C09113=1137.061,-43.555,-47.132,179.183,6.181,149.357
C09114=1137.056,-43.306,-47.143,179.186,6.182,149.356
C09115=1137.051,-43.056,-47.155,179.188,6.183,149.355
C09116=1137.046,-42.806,-47.166,179.191,6.183,149.355
C09117=1137.041,-42.556,-47.177,179.193,6.184,149.354
C09118=1137.035,-42.307,-47.188,179.195,6.184,149.354
C09119=1137.030,-42.057,-47.199,179.198,6.185,149.353
C09120=1137.025,-41.807,-47.211,179.200,6.186,149.353
C09121=1137.020,-41.558,-47.222,179.202,6.186,149.352
C09122=1137.014,-41.308,-47.233,179.205,6.187,149.352
C09123=1137.009,-41.058,-47.245,179.207,6.188,149.351
C09124=1137.004,-40.808,-47.256,179.209,6.189,149.351
C09125=1136.998,-40.559,-47.267,179.212,6.189,149.350
C09126=1136.994,-40.309,-47.279,179.214,6.190,149.350
C09127=1136.988,-40.060,-47.291,179.216,6.191,149.349
C09128=1136.984,-39.810,-47.302,179.219,6.191,149.348
C09129=1136.977,-39.560,-47.313,179.221,6.192,149.348
C09130=1136.973,-39.310,-47.324,179.223,6.193,149.347
C09131=1136.967,-39.060,-47.336,179.226,6.193,149.347
C09132=1136.962,-38.811,-47.347,179.228,6.194,149.346
C09133=1136.956,-38.562,-47.359,179.230,6.195,149.346
C09134=1136.952,-38.312,-47.370,179.233,6.195,149.345
C09135=1136.946,-38.062,-47.382,179.235,6.196,149.345
C09136=1136.942,-37.812,-47.393,179.237,6.196,149.344
C09137=1136.936,-37.563,-47.405,179.239,6.196,149.343
C09138=1136.930,-37.313,-47.416,179.241,6.197,149.343
C09139=1136.925,-37.063,-47.427,179.244,6.198,149.342
C09140=1136.920,-36.813,-47.439,179.246,6.198,149.342
C09141=1136.915,-36.563,-47.450,179.248,6.199,149.341
C09142=1136.909,-36.314,-47.462,179.251,6.200,149.341
C09143=1136.904,-36.065,-47.473,179.253,6.200,149.340
C09144=1136.899,-35.815,-47.485,179.255,6.201,149.340
C09145=1136.893,-35.565,-47.497,179.258,6.202,149.339
C09146=1136.889,-35.315,-47.508,179.260,6.202,149.339
C09147=1136.883,-35.066,-47.520,179.263,6.203,149.338
C09148=1136.878,-34.816,-47.531,179.265,6.204,149.337
C09149=1136.873,-34.566,-47.543,179.267,6.204,149.337
C09150=1136.868,-34.317,-47.554,179.270,6.205,149.336
C09151=1136.862,-34.067,-47.566,179.272,6.206,149.336
C09152=1136.857,-33.817,-47.578,179.274,6.206,149.335
C09153=1136.852,-33.568,-47.589,179.277,6.207,149.335
C09154=1136.847,-33.319,-47.601,179.279,6.208,149.334
C09155=1136.841,-33.069,-47.613,179.281,6.208,149.334
C09156=1136.836,-32.819,-47.625,179.284,6.209,149.333
C09157=1136.831,-32.569,-47.637,179.286,6.210,149.333
C09158=1136.826,-32.319,-47.648,179.288,6.210,149.332
C09159=1136.821,-32.069,-47.660,179.291,6.211,149.331
C09160=1136.815,-31.820,-47.671,179.293,6.212,149.331
C09161=1136.810,-31.571,-47.683,179.296,6.213,149.330
C09162=1136.805,-31.321,-47.694,179.298,6.213,149.330
C09163=1136.799,-31.071,-47.706,179.301,6.214,149.329
C09164=1136.794,-30.821,-47.719,179.303,6.215,149.329
C09165=1136.790,-30.572,-47.730,179.305,6.215,149.328
C09166=1136.784,-30.322,-47.742,179.308,6.216,149.328
C09167=1136.779,-30.072,-47.754,179.310,6.217,149.327
C09168=1136.773,-29.823,-47.765,179.312,6.217,149.326
C09169=1136.768,-29.573,-47.777,179.315,6.218,149.326
C09170=1136.763,-29.324,-47.789,179.317,6.219,149.325
C09171=1136.758,-29.074,-47.801,179.319,6.219,149.325
C09172=1136.753,-28.824,-47.813,179.322,6.220,149.324
C09173=1136.747,-28.574,-47.824,179.324,6.221,149.324
C09174=1136.742,-28.324,-47.836,179.326,6.221,149.323
C09175=1136.737,-28.075,-47.848,179.329,6.222,149.323
C09176=1136.732,-27.825,-47.860,179.331,6.223,149.322
C09177=1136.727,-27.575,-47.872,179.333,6.223,149.321
C09178=1136.721,-27.325,-47.884,179.336,6.224,149.321
C09179=1136.717,-27.076,-47.896,179.338,6.225,149.321
C09180=1136.711,-26.827,-47.908,179.341,6.225,149.320
C09181=1136.706,-26.577,-47.920,179.343,6.226,149.319
C09182=1136.701,-26.327,-47.932,179.345,6.227,149.319
C09183=1136.696,-26.078,-47.943,179.348,6.227,149.318
C09184=1136.690,-25.828,-47.955,179.350,6.228,149.318
C09185=1136.685,-25.579,-47.967,179.352,6.229,149.317
C09186=1136.680,-25.329,-47.980,179.355,6.230,149.317
C09187=1136.674,-25.059,-47.993,179.357,6.231,149.316
C09188=1136.669,-24.788,-48.006,179.360,6.231,149.315
C09189=1136.663,-24.519,-48.018,179.362,6.232,149.315
C09190=1136.657,-24.248,-48.032,179.365,6.232,149.314
C09191=1136.653,-23.999,-48.044,179.368,6.234,149.314
C09192=1136.647,-23.749,-48.056,179.370,6.235,149.313
C09193=1136.642,-23.499,-48.067,179.373,6.235,149.313
C09194=1136.637,-23.250,-48.080,179.375,6.236,149.312
C09195=1136.631,-23.000,-48.092,179.377,6.237,149.312
C09196=1136.626,-22.750,-48.104,179.380,6.237,149.311
C09197=1136.621,-22.501,-48.116,179.382,6.238,149.310
C09198=1136.616,-22.251,-48.128,179.384,6.238,149.310
C09199=1136.611,-22.002,-48.140,179.387,6.239,149.309
C09200=1136.605,-21.752,-48.152,179.389,6.240,149.309
C09201=1136.600,-21.503,-48.165,179.391,6.240,149.308
C09202=1136.595,-21.253,-48.177,179.394,6.241,149.308
C09203=1136.589,-21.003,-48.189,179.396,6.242,149.307
C09204=1136.584,-20.753,-48.201,179.399,6.243,149.306
C09205=1136.579,-20.503,-48.213,179.401,6.244,149.306
C09206=1136.574,-20.254,-48.226,179.403,6.245,149.306
C09207=1136.568,-20.004,-48.238,179.406,6.245,149.305
C09208=1136.563,-19.755,-48.250,179.408,6.246,149.304
C09209=1136.558,-19.505,-48.262,179.410,6.247,149.304
C09210=1136.553,-19.256,-48.275,179.413,6.247,149.303
C09211=1136.547,-19.006,-48.287,179.415,6.248,149.303
C09212=1136.543,-18.756,-48.299,179.417,6.249,149.302
C09213=1136.538,-18.507,-48.312,179.420,6.249,149.302
C09214=1136.533,-18.257,-48.323,179.422,6.250,149.301
C09215=1136.528,-18.007,-48.336,179.425,6.252,149.301
C09216=1136.522,-17.757,-48.348,179.428,6.252,149.300
C09217=1136.517,-17.508,-48.360,179.430,6.253,149.299
C09218=1136.512,-17.258,-48.372,179.432,6.254,149.299
C09219=1136.507,-17.009,-48.385,179.435,6.254,149.298
C09220=1136.501,-16.760,-48.398,179.437,6.255,149.298
C09221=1136.496,-16.510,-48.409,179.439,6.256,149.297
C09222=1136.491,-16.260,-48.422,179.442,6.256,149.297
C09223=1136.486,-16.010,-48.434,179.444,6.257,149.296
C09224=1136.481,-15.760,-48.447,179.447,6.258,149.296
C09225=1136.475,-15.511,-48.460,179.449,6.259,149.295
C09226=1136.470,-15.261,-48.472,179.452,6.259,149.295
C09227=1136.465,-15.011,-48.485,179.454,6.260,149.294
C09228=1136.459,-14.762,-48.497,179.456,6.261,149.293
C09229=1136.454,-14.512,-48.509,179.459,6.261,149.293
C09230=1136.449,-14.263,-48.522,179.461,6.262,149.292
C09231=1136.444,-14.013,-48.535,179.463,6.263,149.292
C09232=1136.439,-13.763,-48.547,179.466,6.264,149.291
C09233=1136.434,-13.514,-48.559,179.469,6.265,149.291
C09234=1136.429,-13.264,-48.572,179.471,6.265,149.290
C09235=1136.424,-13.015,-48.584,179.473,6.266,149.290
C09236=1136.418,-12.765,-48.596,179.476,6.267,149.289
C09237=1136.414,-12.515,-48.609,179.478,6.267,149.288
C09238=1136.408,-12.265,-48.622,179.480,6.268,149.288
C09239=1136.403,-12.016,-48.635,179.484,6.269,149.287
C09240=1136.397,-11.766,-48.647,179.486,6.270,149.287
C09241=1136.392,-11.517,-48.659,179.488,6.271,149.286
C09242=1136.388,-11.267,-48.672,179.491,6.271,149.286
C09243=1136.382,-11.018,-48.685,179.493,6.272,149.285
C09244=1136.377,-10.768,-48.698,179.495,6.273,149.285
C09245=1136.372,-10.518,-48.710,179.498,6.274,149.284
C09246=1136.366,-10.269,-48.723,179.500,6.275,149.284
C09247=1136.361,-10.019,-48.736,179.503,6.276,149.283
C09248=1136.356,-9.769,-48.748,179.505,6.276,149.282
C09249=1136.351,-9.520,-48.761,179.507,6.277,149.282
C09250=1136.346,-9.271,-48.773,179.510,6.278,149.281
C09251=1136.341,-9.020,-48.786,179.512,6.278,149.281
C09252=1136.335,-8.770,-48.799,179.515,6.280,149.280
C09253=1136.330,-8.521,-48.812,179.518,6.280,149.280
C09254=1136.325,-8.272,-48.824,179.520,6.281,149.279
C09255=1136.320,-8.022,-48.837,179.522,6.282,149.279
C09256=1136.316,-7.772,-48.850,179.525,6.282,149.278
C09257=1136.310,-7.523,-48.863,179.527,6.283,149.278
C09258=1136.305,-7.273,-48.876,179.530,6.285,149.277
C09259=1136.299,-7.024,-48.888,179.532,6.285,149.276
C09260=1136.295,-6.774,-48.901,179.534,6.286,149.276
C09261=1136.289,-6.524,-48.914,179.537,6.287,149.275
C09262=1136.284,-6.275,-48.926,179.539,6.287,149.275
C09263=1136.279,-6.025,-48.939,179.542,6.289,149.274
C09264=1136.274,-5.775,-48.952,179.544,6.290,149.274
C09265=1136.268,-5.526,-48.965,179.547,6.290,149.273
C09266=1136.263,-5.276,-48.978,179.549,6.291,149.273
C09267=1136.258,-5.026,-48.990,179.552,6.291,149.272
C09268=1136.253,-4.777,-49.004,179.554,6.292,149.272
C09269=1136.247,-4.527,-49.016,179.557,6.294,149.271
C09270=1136.243,-4.277,-49.029,179.559,6.294,149.270
C09271=1136.237,-4.028,-49.042,179.562,6.295,149.270
C09272=1136.232,-3.778,-49.055,179.564,6.296,149.269
C09273=1136.227,-3.528,-49.068,179.566,6.296,149.269
C09274=1136.222,-3.279,-49.082,179.569,6.298,149.268
C09275=1136.217,-3.030,-49.095,179.571,6.298,149.268
C09276=1136.212,-2.780,-49.107,179.574,6.299,149.267
C09277=1136.206,-2.530,-49.121,179.576,6.300,149.267
C09278=1136.201,-2.281,-49.133,179.578,6.300,149.266
C09279=1136.197,-2.031,-49.146,179.582,6.302,149.265
C09280=1136.191,-1.781,-49.159,179.584,6.302,149.265
C09281=1136.186,-1.532,-49.172,179.586,6.303,149.265
C09282=1136.181,-1.282,-49.185,179.589,6.304,149.264
C09283=1136.175,-1.032,-49.198,179.591,6.305,149.263
C09284=1136.171,-0.784,-49.212,179.594,6.306,149.263
C09285=1136.165,-0.533,-49.225,179.596,6.307,149.262
C09286=1136.160,-0.284,-49.238,179.598,6.307,149.262
C09287=1136.155,-0.035,-49.250,179.601,6.308,149.261
C09288=1136.150,0.216,-49.264,179.604,6.309,149.261
C09289=1136.145,0.465,-49.276,179.606,6.310,149.260
C09290=1136.140,0.715,-49.291,179.609,6.311,149.259
C09291=1136.134,0.984,-49.304,179.611,6.312,149.259
C09292=1136.128,1.254,-49.318,179.614,6.313,149.258
C09293=1136.123,1.523,-49.333,179.616,6.313,149.258
C09294=1136.117,1.792,-49.347,179.620,6.315,149.257
C09295=1136.112,2.042,-49.360,179.622,6.315,149.257
C09296=1136.107,2.291,-49.374,179.624,6.316,149.256
C09297=1136.102,2.541,-49.387,179.627,6.317,149.256
C09298=1136.097,2.791,-49.400,179.629,6.318,149.255
C09299=1136.091,3.040,-49.413,179.632,6.319,149.254
C09300=1136.087,3.290,-49.427,179.634,6.319,149.254
C09301=1136.081,3.539,-49.440,179.636,6.320,149.253
C09302=1136.076,3.789,-49.453,179.640,6.321,149.253
C09303=1136.071,4.038,-49.467,179.642,6.322,149.252
C09304=1136.066,4.288,-49.480,179.644,6.323,149.252
C09305=1136.060,4.538,-49.493,179.647,6.324,149.251
C09306=1136.056,4.787,-49.506,179.649,6.325,149.251
C09307=1136.050,5.037,-49.520,179.652,6.326,149.250
C09308=1136.045,5.286,-49.532,179.654,6.326,149.250
C09309=1136.040,5.536,-49.547,179.656,6.327,149.249
C09310=1136.035,5.785,-49.559,179.659,6.329,149.249
C09311=1136.030,6.036,-49.573,179.662,6.329,149.248
C09312=1136.024,6.285,-49.587,179.664,6.330,149.247
C09313=1136.020,6.535,-49.600,179.667,6.331,149.247
C09314=1136.014,6.784,-49.613,179.669,6.332,149.246
C09315=1136.010,7.034,-49.626,179.672,6.333,149.246
C09316=1136.004,7.283,-49.640,179.674,6.333,149.245
C09317=1136.000,7.533,-49.653,179.677,6.335,149.245
C09318=1135.994,7.782,-49.667,179.679,6.336,149.244
C09319=1135.989,8.032,-49.681,179.682,6.336,149.244
C09320=1135.984,8.282,-49.693,179.684,6.337,149.243
C09321=1135.979,8.531,-49.708,179.687,6.338,149.243
C09322=1135.973,8.781,-49.721,179.689,6.339,149.242
C09323=1135.969,9.030,-49.735,179.692,6.340,149.241
C09324=1135.963,9.280,-49.748,179.694,6.341,149.241
C09325=1135.959,9.529,-49.761,179.697,6.342,149.240
C09326=1135.953,9.780,-49.775,179.699,6.343,149.240
C09327=1135.948,10.029,-49.789,179.701,6.343,149.239
C09328=1135.943,10.279,-49.802,179.705,6.345,149.239
C09329=1135.938,10.528,-49.816,179.707,6.345,149.238
C09330=1135.932,10.778,-49.829,179.710,6.346,149.238
C09331=1135.928,11.027,-49.843,179.712,6.347,149.237
C09332=1135.922,11.277,-49.856,179.714,6.348,149.237
C09333=1135.917,11.526,-49.870,179.717,6.349,149.236
C09334=1135.912,11.776,-49.884,179.719,6.349,149.236
C09335=1135.907,12.026,-49.897,179.722,6.351,149.235
C09336=1135.902,12.275,-49.911,179.725,6.352,149.234
C09337=1135.897,12.525,-49.925,179.727,6.352,149.234
C09338=1135.892,12.774,-49.938,179.730,6.354,149.233
C09339=1135.887,13.024,-49.952,179.732,6.354,149.233
C09340=1135.881,13.273,-49.966,179.735,6.355,149.232
C09341=1135.876,13.523,-49.980,179.737,6.357,149.232
C09342=1135.872,13.772,-49.994,179.740,6.357,149.231
C09343=1135.866,14.022,-50.007,179.742,6.358,149.231
C09344=1135.861,14.272,-50.021,179.745,6.360,149.230
C09345=1135.856,14.521,-50.035,179.748,6.360,149.230
C09346=1135.851,14.771,-50.048,179.750,6.361,149.229
C09347=1135.846,15.020,-50.062,179.752,6.363,149.229
C09348=1135.840,15.269,-50.076,179.755,6.363,149.228
C09349=1135.835,15.520,-50.090,179.757,6.364,149.227
C09350=1135.830,15.769,-50.104,179.761,6.365,149.227
C09351=1135.825,16.018,-50.117,179.763,6.366,149.226
C09352=1135.820,16.268,-50.132,179.765,6.367,149.226
C09353=1135.815,16.518,-50.145,179.768,6.368,149.225
C09354=1135.809,16.767,-50.159,179.770,6.369,149.225
C09355=1135.805,17.017,-50.173,179.772,6.369,149.224
C09356=1135.800,17.267,-50.188,179.776,6.371,149.224
C09357=1135.794,17.516,-50.200,179.778,6.372,149.223
C09358=1135.790,17.766,-50.214,179.780,6.372,149.223
C09359=1135.785,18.015,-50.229,179.783,6.374,149.222
C09360=1135.779,18.264,-50.243,179.786,6.374,149.222
C09361=1135.774,18.514,-50.257,179.788,6.375,149.221
C09362=1135.769,18.764,-50.271,179.791,6.376,149.220
C09363=1135.763,19.013,-50.284,179.793,6.377,149.220
C09364=1135.758,19.263,-50.299,179.795,6.378,149.219
C09365=1135.754,19.512,-50.312,179.799,6.379,149.219
C09366=1135.749,19.761,-50.326,179.801,6.380,149.218
C09367=1135.744,20.011,-50.341,179.803,6.381,149.218
C09368=1135.739,20.261,-50.355,179.806,6.382,149.217
C09369=1135.734,20.511,-50.369,179.808,6.383,149.217
C09370=1135.728,20.760,-50.383,179.811,6.385,149.216
C09371=1135.723,21.009,-50.397,179.814,6.385,149.216
C09372=1135.718,21.260,-50.411,179.816,6.386,149.215
C09373=1135.713,21.509,-50.425,179.819,6.387,149.215
C09374=1135.707,21.758,-50.439,179.821,6.388,149.214
C09375=1135.702,22.008,-50.453,179.823,6.389,149.214
C09376=1135.697,22.258,-50.468,179.827,6.390,149.213
C09377=1135.692,22.508,-50.482,179.829,6.391,149.212
C09378=1135.687,22.757,-50.496,179.831,6.392,149.212
C09379=1135.682,23.006,-50.510,179.834,6.393,149.211
C09380=1135.677,23.256,-50.524,179.836,6.394,149.211
C09381=1135.672,23.506,-50.539,179.839,6.395,149.210
C09382=1135.667,23.755,-50.553,179.842,6.396,149.210
C09383=1135.662,24.004,-50.567,179.844,6.396,149.209
C09384=1135.657,24.254,-50.581,179.847,6.398,149.209
C09385=1135.652,24.504,-50.595,179.849,6.399,149.208
C09386=1135.647,24.753,-50.610,179.852,6.400,149.208
C09387=1135.641,25.002,-50.624,179.854,6.401,149.207
C09388=1135.636,25.252,-50.639,179.857,6.401,149.206
C09389=1135.632,25.501,-50.653,179.860,6.403,149.206
C09390=1135.627,25.751,-50.667,179.862,6.404,149.206
C09391=1135.622,26.001,-50.681,179.865,6.405,149.205
C09392=1135.616,26.250,-50.695,179.867,6.406,149.204
C09393=1135.611,26.499,-50.710,179.870,6.407,149.204
C09394=1135.606,26.749,-50.724,179.873,6.408,149.203
C09395=1135.600,27.018,-50.740,179.875,6.409,149.203
C09396=1135.595,27.288,-50.755,179.878,6.410,149.202
C09397=1135.590,27.556,-50.771,179.881,6.412,149.202
C09398=1135.584,27.825,-50.786,179.884,6.412,149.201
C09399=1135.579,28.074,-50.800,179.886,6.414,149.201
C09400=1135.574,28.324,-50.815,179.889,6.415,149.200
C09401=1135.568,28.574,-50.830,179.891,6.415,149.199
C09402=1135.563,28.824,-50.844,179.894,6.417,149.199
C09403=1135.559,29.073,-50.859,179.896,6.417,149.199
C09404=1135.554,29.323,-50.873,179.899,6.419,149.198
C09405=1135.549,29.572,-50.887,179.902,6.419,149.197
C09406=1135.543,29.821,-50.901,179.904,6.421,149.197
C09407=1135.538,30.071,-50.917,179.907,6.422,149.196
C09408=1135.533,30.320,-50.931,179.909,6.422,149.196
C09409=1135.528,30.570,-50.946,179.912,6.424,149.195
C09410=1135.523,30.820,-50.960,179.915,6.424,149.195
C09411=1135.518,31.069,-50.975,179.917,6.426,149.194
C09412=1135.513,31.319,-50.989,179.920,6.427,149.194
C09413=1135.508,31.569,-51.004,179.923,6.428,149.193
C09414=1135.503,31.818,-51.019,179.925,6.429,149.193
C09415=1135.498,32.067,-51.033,179.927,6.430,149.192
C09416=1135.493,32.316,-51.047,179.930,6.431,149.192
C09417=1135.487,32.566,-51.063,179.933,6.432,149.191
C09418=1135.482,32.816,-51.077,179.935,6.433,149.191
C09419=1135.477,33.065,-51.091,179.938,6.434,149.190
C09420=1135.473,33.314,-51.106,179.941,6.435,149.189
C09421=1135.467,33.564,-51.121,179.943,6.436,149.189
C09422=1135.462,33.813,-51.136,179.946,6.438,149.188
C09423=1135.457,34.063,-51.150,179.948,6.438,149.188
C09424=1135.452,34.313,-51.165,179.951,6.440,149.187
C09425=1135.447,34.562,-51.180,179.954,6.440,149.187
C09426=1135.442,34.812,-51.195,179.956,6.441,149.186
C09427=1135.437,35.061,-51.210,179.959,6.443,149.186
C09428=1135.432,35.311,-51.224,179.961,6.443,149.185
C09429=1135.427,35.560,-51.239,179.964,6.445,149.185
C09430=1135.422,35.810,-51.254,179.966,6.446,149.184
C09431=1135.417,36.059,-51.269,179.969,6.447,149.184
C09432=1135.412,36.309,-51.284,179.972,6.448,149.183
C09433=1135.407,36.558,-51.299,179.974,6.449,149.183
C09434=1135.401,36.808,-51.313,179.977,6.450,149.182
C09435=1135.397,37.057,-51.328,179.980,6.452,149.182
C09436=1135.392,37.307,-51.343,179.982,6.452,149.181
C09437=1135.386,37.556,-51.358,179.985,6.454,149.180
C09438=1135.382,37.806,-51.373,179.987,6.454,149.180
C09439=1135.376,38.055,-51.388,179.990,6.456,149.180
C09440=1135.371,38.305,-51.402,179.993,6.457,149.179
C09441=1135.367,38.554,-51.417,179.996,6.458,149.178
C09442=1135.361,38.804,-51.432,179.998,6.459,149.178
C09443=1135.356,39.053,-51.447,-180.000,6.461,149.178
C09444=1135.351,39.303,-51.463,-179.997,6.461,149.177
C09445=1135.346,39.552,-51.477,-179.994,6.463,149.176
C09446=1135.340,39.802,-51.493,-179.992,6.464,149.176
C09447=1135.335,40.052,-51.507,-179.989,6.465,149.175
C09448=1135.331,40.301,-51.522,-179.987,6.466,149.175
C09449=1135.325,40.550,-51.538,-179.984,6.467,149.174
C09450=1135.321,40.800,-51.552,-179.981,6.468,149.174
C09451=1135.315,41.049,-51.567,-179.978,6.469,149.173
C09452=1135.311,41.299,-51.583,-179.976,6.470,149.173
C09453=1135.305,41.549,-51.598,-179.973,6.471,149.172
C09454=1135.301,41.798,-51.613,-179.971,6.472,149.172
C09455=1135.295,42.047,-51.628,-179.968,6.474,149.171
C09456=1135.291,42.297,-51.643,-179.965,6.474,149.171
C09457=1135.285,42.547,-51.658,-179.963,6.476,149.170
C09458=1135.280,42.796,-51.673,-179.960,6.477,149.170
C09459=1135.275,43.045,-51.689,-179.958,6.478,149.169
C09460=1135.270,43.294,-51.704,-179.955,6.479,149.169
C09461=1135.265,43.545,-51.719,-179.952,6.480,149.168
C09462=1135.261,43.794,-51.734,-179.950,6.481,149.168
C09463=1135.255,44.043,-51.749,-179.947,6.483,149.167
C09464=1135.251,44.292,-51.764,-179.945,6.483,149.167
C09465=1135.245,44.542,-51.779,-179.942,6.485,149.166
C09466=1135.239,44.792,-51.795,-179.939,6.485,149.165
C09467=1135.235,45.041,-51.810,-179.937,6.487,149.165
C09468=1135.230,45.291,-51.826,-179.934,6.489,149.165
C09469=1135.225,45.540,-51.841,-179.931,6.489,149.164
C09470=1135.220,45.790,-51.856,-179.928,6.491,149.163
C09471=1135.215,46.039,-51.871,-179.926,6.492,149.163
C09472=1135.210,46.289,-51.886,-179.923,6.493,149.163
C09473=1135.204,46.538,-51.902,-179.921,6.494,149.162
C09474=1135.200,46.788,-51.917,-179.918,6.495,149.161
C09475=1135.195,47.037,-51.933,-179.916,6.496,149.161
C09476=1135.190,47.286,-51.948,-179.913,6.497,149.160
C09477=1135.185,47.536,-51.963,-179.911,6.498,149.160
C09478=1135.179,47.785,-51.979,-179.908,6.500,149.159
C09479=1135.175,48.035,-51.994,-179.905,6.501,149.159
C09480=1135.170,48.284,-52.010,-179.902,6.502,149.158
C09481=1135.165,48.534,-52.026,-179.900,6.504,149.158
C09482=1135.160,48.783,-52.041,-179.897,6.504,149.157
C09483=1135.155,49.032,-52.056,-179.894,6.506,149.157
C09484=1135.150,49.282,-52.072,-179.892,6.507,149.156
C09485=1135.145,49.531,-52.087,-179.889,6.508,149.156
C09486=1135.140,49.781,-52.103,-179.886,6.509,149.155
C09487=1135.134,50.030,-52.118,-179.884,6.510,149.155
C09488=1135.130,50.280,-52.134,-179.881,6.512,149.154
C09489=1135.125,50.529,-52.149,-179.878,6.512,149.154
C09490=1135.120,50.779,-52.165,-179.876,6.514,149.153
C09491=1135.114,51.028,-52.180,-179.874,6.515,149.153
C09492=1135.110,51.278,-52.196,-179.871,6.516,149.152
C09493=1135.105,51.527,-52.211,-179.868,6.518,149.152
C09494=1135.099,51.777,-52.227,-179.865,6.519,149.151
C09495=1135.094,52.026,-52.243,-179.863,6.520,149.151
C09496=1135.090,52.276,-52.258,-179.860,6.521,149.150
C09497=1135.084,52.525,-52.273,-179.857,6.522,149.150
C09498=1135.079,52.774,-52.290,-179.854,6.524,149.149
C09499=1135.074,53.043,-52.306,-179.852,6.524,149.149
C09500=1135.069,53.313,-52.323,-179.849,6.526,149.148
C09501=1135.063,53.581,-52.340,-179.846,6.527,149.147
C09502=1135.058,53.849,-52.357,-179.843,6.529,149.147
C09503=1135.053,54.099,-52.372,-179.841,6.530,149.147
C09504=1135.048,54.349,-52.388,-179.838,6.531,149.146
C09505=1135.043,54.597,-52.405,-179.835,6.533,149.145
C09506=1135.038,54.847,-52.420,-179.833,6.533,149.145
C09507=1135.033,55.097,-52.436,-179.830,6.535,149.145
C09508=1135.027,55.346,-52.452,-179.827,6.536,149.144
C09509=1135.023,55.595,-52.467,-179.825,6.537,149.143
C09510=1135.018,55.845,-52.484,-179.822,6.539,149.143
C09511=1135.013,56.094,-52.499,-179.819,6.539,149.142
C09512=1135.007,56.344,-52.515,-179.816,6.541,149.142
C09513=1135.003,56.594,-52.531,-179.814,6.542,149.141
C09514=1134.998,56.843,-52.547,-179.812,6.543,149.141
C09515=1134.992,57.092,-52.563,-179.808,6.545,149.140
C09516=1134.987,57.342,-52.579,-179.806,6.546,149.140
C09517=1134.982,57.591,-52.595,-179.803,6.547,149.139
C09518=1134.978,57.840,-52.610,-179.801,6.549,149.139
C09519=1134.973,58.090,-52.626,-179.798,6.549,149.138
C09520=1134.968,58.339,-52.642,-179.795,6.551,149.138
C09521=1134.963,58.589,-52.658,-179.792,6.553,149.137
C09522=1134.958,58.838,-52.674,-179.790,6.553,149.137
C09523=1134.953,59.087,-52.690,-179.787,6.555,149.136
C09524=1134.948,59.337,-52.706,-179.785,6.556,149.136
C09525=1134.943,59.586,-52.722,-179.782,6.557,149.135
C09526=1134.938,59.836,-52.738,-179.779,6.558,149.135
C09527=1134.933,60.086,-52.754,-179.777,6.559,149.134
C09528=1134.928,60.335,-52.770,-179.774,6.561,149.134
C09529=1134.923,60.584,-52.786,-179.771,6.563,149.133
C09530=1134.918,60.833,-52.802,-179.769,6.563,149.133
C09531=1134.913,61.083,-52.818,-179.766,6.565,149.132
C09532=1134.908,61.332,-52.835,-179.763,6.566,149.132
C09533=1134.903,61.582,-52.850,-179.761,6.567,149.131
C09534=1134.898,61.831,-52.867,-179.758,6.568,149.131
C09535=1134.893,62.081,-52.883,-179.755,6.570,149.130
C09536=1134.888,62.330,-52.899,-179.753,6.571,149.130
C09537=1134.883,62.580,-52.915,-179.750,6.572,149.129
C09538=1134.878,62.829,-52.931,-179.747,6.574,149.129
C09539=1134.873,63.079,-52.947,-179.745,6.575,149.128
C09540=1134.868,63.328,-52.964,-179.742,6.576,149.128
C09541=1134.863,63.578,-52.980,-179.739,6.578,149.127
C09542=1134.858,63.827,-52.996,-179.737,6.578,149.127
C09543=1134.853,64.077,-53.012,-179.734,6.580,149.126
C09544=1134.848,64.326,-53.029,-179.731,6.582,149.126
C09545=1134.843,64.575,-53.045,-179.728,6.582,149.125
C09546=1134.838,64.825,-53.061,-179.726,6.584,149.125
C09547=1134.833,65.074,-53.078,-179.723,6.585,149.124
C09548=1134.828,65.323,-53.094,-179.721,6.586,149.124
C09549=1134.824,65.573,-53.110,-179.718,6.588,149.123
C09550=1134.819,65.822,-53.126,-179.715,6.589,149.123
C09551=1134.813,66.072,-53.143,-179.713,6.590,149.123
C09552=1134.808,66.321,-53.159,-179.710,6.592,149.122
C09553=1134.803,66.571,-53.176,-179.707,6.593,149.121
C09554=1134.798,66.819,-53.192,-179.704,6.595,149.121
C09555=1134.794,67.069,-53.208,-179.702,6.595,149.121
C09556=1134.788,67.318,-53.224,-179.699,6.597,149.120
C09557=1134.783,67.568,-53.241,-179.696,6.598,149.119
C09558=1134.778,67.818,-53.257,-179.694,6.599,149.119
C09559=1134.773,68.067,-53.274,-179.691,6.601,149.119
C09560=1134.769,68.316,-53.290,-179.688,6.602,149.118
C09561=1134.764,68.565,-53.307,-179.685,6.603,149.117
C09562=1134.758,68.816,-53.323,-179.683,6.605,149.117
C09563=1134.754,69.065,-53.340,-179.680,6.606,149.117
C09564=1134.749,69.314,-53.356,-179.677,6.608,149.116
C09565=1134.744,69.563,-53.373,-179.675,6.608,149.116
C09566=1134.738,69.812,-53.390,-179.672,6.610,149.115
C09567=1134.734,70.062,-53.406,-179.669,6.612,149.115
C09568=1134.729,70.312,-53.422,-179.666,6.613,149.114
C09569=1134.724,70.561,-53.439,-179.664,6.614,149.114
C09570=1134.719,70.811,-53.456,-179.661,6.615,149.113
C09571=1134.714,71.059,-53.472,-179.658,6.617,149.113
C09572=1134.709,71.309,-53.489,-179.656,6.618,149.112
C09573=1134.704,71.559,-53.506,-179.653,6.620,149.112
C09574=1134.699,71.808,-53.522,-179.650,6.621,149.111
C09575=1134.694,72.057,-53.538,-179.647,6.623,149.111
C09576=1134.689,72.307,-53.556,-179.645,6.623,149.110
C09577=1134.684,72.556,-53.572,-179.642,6.625,149.110
C09578=1134.679,72.806,-53.589,-179.639,6.626,149.109
C09579=1134.674,73.055,-53.606,-179.636,6.628,149.109
C09580=1134.669,73.304,-53.622,-179.634,6.629,149.108
C09581=1134.665,73.554,-53.639,-179.631,6.630,149.108
C09582=1134.659,73.803,-53.656,-179.629,6.632,149.107
C09583=1134.654,74.052,-53.673,-179.626,6.633,149.107
C09584=1134.650,74.302,-53.689,-179.623,6.634,149.106
C09585=1134.645,74.551,-53.706,-179.621,6.636,149.106
C09586=1134.640,74.800,-53.723,-179.618,6.638,149.106
C09587=1134.634,75.050,-53.740,-179.615,6.639,149.105
C09588=1134.630,75.300,-53.757,-179.612,6.640,149.104
C09589=1134.625,75.549,-53.773,-179.610,6.641,149.104
C09590=1134.620,75.798,-53.790,-179.607,6.643,149.104
C09591=1134.615,76.048,-53.807,-179.604,6.645,149.103
C09592=1134.610,76.297,-53.824,-179.602,6.645,149.103
C09593=1134.605,76.546,-53.841,-179.599,6.647,149.102
C09594=1134.600,76.796,-53.858,-179.596,6.648,149.102
C09595=1134.595,77.045,-53.875,-179.593,6.650,149.101
C09596=1134.590,77.295,-53.892,-179.591,6.652,149.101
C09597=1134.585,77.543,-53.909,-179.588,6.652,149.100
C09598=1134.580,77.793,-53.926,-179.585,6.654,149.100
C09599=1134.575,78.043,-53.943,-179.582,6.655,149.099
C09600=1134.570,78.293,-53.960,-179.580,6.657,149.099
C09601=1134.565,78.541,-53.976,-179.578,6.658,149.098
C09602=1134.560,78.790,-53.994,-179.574,6.659,149.098
C09603=1134.556,79.059,-54.012,-179.572,6.661,149.097
C09604=1134.550,79.327,-54.031,-179.569,6.663,149.097
C09605=1134.545,79.596,-54.049,-179.566,6.664,149.096
C09606=1134.540,79.865,-54.067,-179.563,6.666,149.096
C09607=1134.534,80.114,-54.084,-179.560,6.667,149.095
C09608=1134.529,80.363,-54.101,-179.557,6.668,149.095
C09609=1134.524,80.612,-54.119,-179.554,6.670,149.094
C09610=1134.520,80.862,-54.136,-179.552,6.671,149.094
C09611=1134.515,81.112,-54.153,-179.549,6.673,149.093
C09612=1134.510,81.360,-54.170,-179.547,6.674,149.093
C09613=1134.505,81.610,-54.187,-179.543,6.676,149.092
C09614=1134.499,81.859,-54.204,-179.541,6.677,149.092
C09615=1134.495,82.109,-54.221,-179.538,6.679,149.092
C09616=1134.490,82.358,-54.239,-179.536,6.680,149.091
C09617=1134.486,82.608,-54.256,-179.533,6.681,149.091
C09618=1134.480,82.856,-54.273,-179.530,6.683,149.090
C09619=1134.475,83.106,-54.291,-179.527,6.684,149.090
C09620=1134.470,83.355,-54.307,-179.524,6.686,149.089
C09621=1134.465,83.604,-54.325,-179.522,6.687,149.089
C09622=1134.460,83.854,-54.343,-179.519,6.688,149.088
C09623=1134.456,84.104,-54.359,-179.517,6.690,149.088
C09624=1134.451,84.353,-54.377,-179.513,6.691,149.087
C09625=1134.446,84.603,-54.394,-179.511,6.693,149.087
C09626=1134.441,84.851,-54.411,-179.508,6.695,149.086
C09627=1134.436,85.101,-54.429,-179.506,6.696,149.086
C09628=1134.431,85.350,-54.447,-179.503,6.697,149.086
C09629=1134.426,85.599,-54.463,-179.500,6.699,149.085
C09630=1134.421,85.849,-54.481,-179.497,6.700,149.084
C09631=1134.416,86.098,-54.499,-179.494,6.702,149.084
C09632=1134.411,86.347,-54.517,-179.492,6.704,149.084
C09633=1134.407,86.597,-54.533,-179.489,6.704,149.083
C09634=1134.402,86.846,-54.551,-179.487,6.706,149.083
C09635=1134.397,87.096,-54.569,-179.483,6.707,149.082
C09636=1134.392,87.345,-54.587,-179.481,6.709,149.082
C09637=1134.387,87.595,-54.603,-179.478,6.711,149.081
C09638=1134.382,87.844,-54.621,-179.475,6.712,149.081
C09639=1134.376,88.093,-54.638,-179.472,6.714,149.080
C09640=1134.372,88.342,-54.656,-179.470,6.715,149.080
C09641=1134.367,88.591,-54.674,-179.467,6.716,149.079
C09642=1134.362,88.841,-54.691,-179.464,6.718,149.079
C09643=1134.357,89.090,-54.709,-179.462,6.719,149.079
C09644=1134.352,89.340,-54.726,-179.459,6.721,149.078
C09645=1134.347,89.589,-54.744,-179.456,6.723,149.078
C09646=1134.342,89.838,-54.762,-179.453,6.724,149.077
C09647=1134.337,90.088,-54.779,-179.451,6.726,149.077
C09648=1134.333,90.337,-54.797,-179.448,6.727,149.076
C09649=1134.328,90.586,-54.815,-179.445,6.728,149.076
C09650=1134.323,90.836,-54.832,-179.442,6.730,149.075
C09651=1134.318,91.085,-54.850,-179.440,6.732,149.075
C09652=1134.313,91.334,-54.868,-179.437,6.733,149.074
C09653=1134.308,91.583,-54.886,-179.434,6.735,149.074
C09654=1134.303,91.833,-54.903,-179.431,6.736,149.073
C09655=1134.299,92.082,-54.920,-179.428,6.738,149.073
C09656=1134.294,92.331,-54.938,-179.426,6.739,149.073
C09657=1134.289,92.580,-54.956,-179.423,6.740,149.072
C09658=1134.284,92.830,-54.974,-179.421,6.742,149.072
C09659=1134.279,93.080,-54.992,-179.418,6.744,149.071
C09660=1134.274,93.329,-55.010,-179.415,6.745,149.071
C09661=1134.269,93.578,-55.028,-179.412,6.747,149.070
C09662=1134.264,93.827,-55.046,-179.409,6.748,149.070
C09663=1134.259,94.077,-55.063,-179.406,6.750,149.069
C09664=1134.254,94.326,-55.081,-179.404,6.752,149.069
C09665=1134.249,94.576,-55.099,-179.401,6.753,149.069
C09666=1134.244,94.825,-55.117,-179.398,6.755,149.068
C09667=1134.240,95.074,-55.135,-179.396,6.756,149.068
C09668=1134.235,95.323,-55.153,-179.393,6.757,149.067
C09669=1134.230,95.572,-55.171,-179.390,6.759,149.067
C09670=1134.225,95.821,-55.189,-179.387,6.760,149.066
C09671=1134.220,96.071,-55.206,-179.385,6.762,149.066
C09672=1134.215,96.321,-55.225,-179.382,6.764,149.065
C09673=1134.210,96.570,-55.243,-179.379,6.765,149.065
C09674=1134.205,96.819,-55.261,-179.376,6.767,149.065
C09675=1134.201,97.069,-55.279,-179.374,6.769,149.064
C09676=1134.196,97.318,-55.297,-179.370,6.770,149.064
C09677=1134.191,97.567,-55.315,-179.368,6.772,149.063
C09678=1134.186,97.816,-55.333,-179.365,6.773,149.063
C09679=1134.181,98.065,-55.350,-179.362,6.775,149.062
C09680=1134.177,98.315,-55.369,-179.360,6.777,149.062
C09681=1134.171,98.565,-55.387,-179.357,6.778,149.061
C09682=1134.166,98.814,-55.405,-179.355,6.779,149.061
C09683=1134.161,99.063,-55.423,-179.352,6.781,149.061
C09684=1134.156,99.312,-55.441,-179.349,6.783,149.060
C09685=1134.152,99.561,-55.460,-179.346,6.784,149.060
C09686=1134.147,99.811,-55.478,-179.343,6.786,149.059
C09687=1134.142,100.060,-55.496,-179.340,6.787,149.059
C09688=1134.138,100.309,-55.514,-179.338,6.789,149.058
C09689=1134.133,100.558,-55.532,-179.335,6.791,149.058
C09690=1134.127,100.808,-55.551,-179.332,6.792,149.057
C09691=1134.123,101.058,-55.569,-179.330,6.794,149.057
C09692=1134.118,101.307,-55.587,-179.327,6.796,149.057
C09693=1134.113,101.556,-55.605,-179.324,6.797,149.056
C09694=1134.108,101.804,-55.624,-179.321,6.799,149.056
C09695=1134.103,102.054,-55.642,-179.318,6.800,149.055
C09696=1134.098,102.304,-55.661,-179.315,6.802,149.055
C09697=1134.093,102.553,-55.679,-179.313,6.804,149.054
C09698=1134.088,102.802,-55.697,-179.310,6.805,149.054
C09699=1134.084,103.051,-55.715,-179.307,6.807,149.053
C09700=1134.079,103.301,-55.734,-179.304,6.809,149.053
C09701=1134.074,103.550,-55.752,-179.302,6.810,149.053
C09702=1134.069,103.799,-55.770,-179.299,6.812,149.052
C09703=1134.064,104.048,-55.789,-179.296,6.814,149.052
C09704=1134.059,104.298,-55.808,-179.293,6.815,149.051
C09705=1134.054,104.547,-55.826,-179.290,6.817,149.051
C09706=1134.050,104.796,-55.845,-179.288,6.818,149.050
C09707=1134.044,105.064,-55.865,-179.285,6.820,149.050
C09708=1134.039,105.333,-55.884,-179.282,6.822,149.050
C09709=1134.034,105.602,-55.904,-179.279,6.823,149.049
C09710=1134.029,105.870,-55.924,-179.276,6.825,149.049
C09711=1134.024,106.119,-55.943,-179.273,6.827,149.048
C09712=1134.019,106.369,-55.962,-179.270,6.829,149.048
C09713=1134.014,106.617,-55.980,-179.267,6.830,149.047
C09714=1134.009,106.867,-55.998,-179.265,6.832,149.047
C09715=1134.004,107.117,-56.017,-179.262,6.834,149.046
C09716=1134.000,107.365,-56.036,-179.259,6.835,149.046
C09717=1133.995,107.614,-56.054,-179.256,6.837,149.046
C09718=1133.990,107.864,-56.073,-179.254,6.839,149.045
C09719=1133.985,108.113,-56.091,-179.251,6.840,149.045
C09720=1133.980,108.362,-56.111,-179.248,6.842,149.044
C09721=1133.976,108.612,-56.129,-179.245,6.844,149.044
C09722=1133.971,108.861,-56.148,-179.243,6.845,149.044
C09723=1133.965,109.110,-56.166,-179.239,6.847,149.043
C09724=1133.961,109.359,-56.185,-179.237,6.848,149.043
C09725=1133.956,109.609,-56.204,-179.234,6.850,149.042
C09726=1133.951,109.857,-56.223,-179.231,6.852,149.042
C09727=1133.946,110.107,-56.242,-179.229,6.853,149.041
C09728=1133.941,110.356,-56.260,-179.226,6.855,149.041
C09729=1133.937,110.606,-56.279,-179.223,6.857,149.040
C09730=1133.932,110.855,-56.298,-179.220,6.858,149.040
C09731=1133.927,111.104,-56.316,-179.218,6.860,149.040
C09732=1133.922,111.354,-56.336,-179.215,6.862,149.039
C09733=1133.917,111.602,-56.354,-179.212,6.864,149.039
C09734=1133.912,111.852,-56.373,-179.209,6.865,149.038
C09735=1133.908,112.101,-56.392,-179.207,6.867,149.038
C09736=1133.902,112.350,-56.410,-179.204,6.869,149.038
C09737=1133.898,112.600,-56.430,-179.201,6.870,149.037
C09738=1133.893,112.848,-56.449,-179.198,6.872,149.037
C09739=1133.888,113.098,-56.467,-179.196,6.874,149.036
C09740=1133.883,113.347,-56.486,-179.193,6.875,149.036
C09741=1133.878,113.597,-56.506,-179.190,6.877,149.036
C09742=1133.873,113.846,-56.524,-179.187,6.879,149.035
C09743=1133.869,114.096,-56.544,-179.184,6.881,149.035
C09744=1133.864,114.344,-56.562,-179.181,6.882,149.034
C09745=1133.859,114.593,-56.582,-179.178,6.884,149.034
C09746=1133.854,114.843,-56.600,-179.176,6.886,149.033
C09747=1133.849,115.092,-56.619,-179.173,6.887,149.033
C09748=1133.844,115.341,-56.639,-179.170,6.889,149.033
C09749=1133.840,115.590,-56.658,-179.167,6.891,149.032
C09750=1133.835,115.839,-56.677,-179.165,6.892,149.032
C09751=1133.829,116.089,-56.696,-179.162,6.894,149.031
C09752=1133.825,116.338,-56.715,-179.159,6.896,149.031
C09753=1133.820,116.587,-56.734,-179.156,6.897,149.030
C09754=1133.816,116.836,-56.753,-179.154,6.899,149.030
C09755=1133.811,117.085,-56.773,-179.151,6.901,149.030
C09756=1133.806,117.335,-56.792,-179.148,6.903,149.029
C09757=1133.801,117.584,-56.810,-179.145,6.905,149.029
C09758=1133.796,117.833,-56.830,-179.142,6.907,149.028
C09759=1133.792,118.083,-56.850,-179.139,6.908,149.028
C09760=1133.786,118.332,-56.869,-179.137,6.910,149.028
C09761=1133.782,118.581,-56.888,-179.134,6.912,149.027
C09762=1133.777,118.830,-56.907,-179.131,6.913,149.027
C09763=1133.772,119.080,-56.927,-179.129,6.915,149.026
C09764=1133.767,119.328,-56.946,-179.126,6.917,149.026
C09765=1133.763,119.578,-56.965,-179.123,6.918,149.026
C09766=1133.757,119.827,-56.985,-179.120,6.921,149.025
C09767=1133.753,120.076,-57.004,-179.117,6.923,149.025
C09768=1133.749,120.325,-57.023,-179.114,6.924,149.024
C09769=1133.743,120.574,-57.043,-179.112,6.926,149.024
C09770=1133.739,120.824,-57.062,-179.109,6.928,149.024
C09771=1133.733,121.073,-57.082,-179.106,6.929,149.023
C09772=1133.729,121.322,-57.101,-179.103,6.931,149.023
C09773=1133.724,121.571,-57.120,-179.101,6.933,149.022
C09774=1133.719,121.820,-57.140,-179.097,6.935,149.022
C09775=1133.714,122.070,-57.159,-179.095,6.937,149.022
C09776=1133.710,122.319,-57.179,-179.092,6.939,149.021
C09777=1133.705,122.568,-57.198,-179.089,6.940,149.021
C09778=1133.700,122.818,-57.217,-179.086,6.942,149.020
C09779=1133.695,123.066,-57.236,-179.084,6.944,149.020
C09780=1133.691,123.315,-57.257,-179.081,6.945,149.020
C09781=1133.686,123.565,-57.277,-179.078,6.947,149.019
C09782=1133.680,123.814,-57.296,-179.075,6.949,149.019
C09783=1133.676,124.063,-57.315,-179.072,6.951,149.018
C09784=1133.672,124.313,-57.335,-179.069,6.953,149.018
C09785=1133.666,124.562,-57.354,-179.067,6.955,149.018
C09786=1133.662,124.810,-57.374,-179.064,6.956,149.017
C09787=1133.657,125.060,-57.394,-179.061,6.958,149.017
C09788=1133.652,125.310,-57.414,-179.059,6.960,149.016
C09789=1133.647,125.559,-57.433,-179.055,6.962,149.016
C09790=1133.643,125.807,-57.453,-179.053,6.964,149.016
C09791=1133.638,126.057,-57.473,-179.050,6.966,149.015
C09792=1133.633,126.306,-57.492,-179.047,6.968,149.015
C09793=1133.628,126.555,-57.512,-179.045,6.969,149.015
C09794=1133.623,126.804,-57.532,-179.042,6.971,149.014
C09795=1133.618,127.053,-57.551,-179.039,6.973,149.014
C09796=1133.614,127.303,-57.570,-179.036,6.975,149.013
C09797=1133.610,127.551,-57.591,-179.033,6.977,149.013
C09798=1133.605,127.801,-57.611,-179.031,6.978,149.013
C09799=1133.599,128.050,-57.630,-179.028,6.980,149.012
C09800=1133.595,128.299,-57.650,-179.025,6.982,149.012
C09801=1133.590,128.548,-57.670,-179.022,6.984,149.011
C09802=1133.585,128.798,-57.690,-179.019,6.986,149.011
C09803=1133.580,129.047,-57.710,-179.016,6.988,149.011
C09804=1133.575,129.296,-57.730,-179.014,6.989,149.010
C09805=1133.571,129.545,-57.750,-179.011,6.991,149.010
C09806=1133.566,129.795,-57.770,-179.008,6.994,149.009
C09807=1133.561,130.044,-57.790,-179.005,6.995,149.009
C09808=1133.556,130.292,-57.809,-179.002,6.997,149.009
C09809=1133.552,130.541,-57.830,-179.000,6.999,149.009
C09810=1133.547,130.791,-57.849,-178.997,7.001,149.008
C09811=1133.542,131.060,-57.871,-178.993,7.003,149.008
C09812=1133.537,131.328,-57.893,-178.991,7.004,149.007
C09813=1133.532,131.597,-57.914,-178.987,7.007,149.007
C09814=1133.526,131.866,-57.936,-178.985,7.009,149.006
C09815=1133.522,132.115,-57.956,-178.982,7.010,149.006
C09816=1133.516,132.363,-57.975,-178.979,7.013,149.006
C09817=1133.512,132.612,-57.996,-178.976,7.015,149.005
C09818=1133.507,132.861,-58.016,-178.974,7.017,149.005
C09819=1133.503,133.111,-58.036,-178.971,7.018,149.005
C09820=1133.497,133.360,-58.057,-178.968,7.020,149.004
C09821=1133.493,133.610,-58.076,-178.965,7.022,149.004
C09822=1133.488,133.858,-58.096,-178.962,7.024,149.003
C09823=1133.483,134.107,-58.117,-178.959,7.026,149.003
C09824=1133.479,134.356,-58.136,-178.957,7.028,149.003
C09825=1133.473,134.606,-58.157,-178.953,7.030,149.002
C09826=1133.469,134.855,-58.178,-178.951,7.032,149.002
C09827=1133.464,135.104,-58.197,-178.948,7.033,149.001
C09828=1133.460,135.353,-58.218,-178.945,7.035,149.001
C09829=1133.455,135.602,-58.238,-178.943,7.037,149.001
C09830=1133.450,135.852,-58.258,-178.940,7.040,149.001
C09831=1133.445,136.100,-58.278,-178.937,7.041,149.000
C09832=1133.440,136.349,-58.299,-178.934,7.043,149.000
C09833=1133.435,136.598,-58.320,-178.931,7.045,148.999
C09834=1133.430,136.848,-58.339,-178.928,7.047,148.999
C09835=1133.426,137.097,-58.360,-178.925,7.049,148.999
C09836=1133.422,137.346,-58.380,-178.923,7.051,148.998
C09837=1133.416,137.595,-58.401,-178.920,7.052,148.998
C09838=1133.412,137.844,-58.422,-178.917,7.055,148.998
C09839=1133.407,138.094,-58.441,-178.914,7.057,148.997
C09840=1133.402,138.343,-58.462,-178.912,7.059,148.997
C09841=1133.398,138.592,-58.483,-178.909,7.060,148.996
C09842=1133.393,138.841,-58.503,-178.906,7.063,148.996
C09843=1133.388,139.090,-58.524,-178.903,7.064,148.996
C09844=1133.384,139.339,-58.544,-178.900,7.066,148.995
C09845=1133.379,139.588,-58.565,-178.897,7.069,148.995
C09846=1133.374,139.838,-58.585,-178.895,7.071,148.995
C09847=1133.369,140.087,-58.605,-178.892,7.072,148.994
C09848=1133.365,140.336,-58.626,-178.889,7.074,148.994
C09849=1133.360,140.585,-58.647,-178.886,7.077,148.994
C09850=1133.355,140.834,-58.667,-178.883,7.078,148.993
C09851=1133.350,141.083,-58.688,-178.880,7.080,148.993
C09852=1133.346,141.332,-58.708,-178.878,7.082,148.992
C09853=1133.341,141.581,-58.729,-178.875,7.085,148.992
C09854=1133.336,141.830,-58.750,-178.872,7.086,148.992
C09855=1133.331,142.079,-58.770,-178.869,7.088,148.991
C09856=1133.326,142.329,-58.791,-178.866,7.090,148.991
C09857=1133.322,142.578,-58.811,-178.863,7.092,148.991
C09858=1133.317,142.827,-58.832,-178.861,7.094,148.990
C09859=1133.312,143.076,-58.853,-178.857,7.096,148.990
C09860=1133.307,143.325,-58.874,-178.855,7.098,148.990
C09861=1133.303,143.574,-58.894,-178.852,7.100,148.989
C09862=1133.298,143.823,-58.916,-178.850,7.102,148.989
C09863=1133.293,144.072,-58.936,-178.846,7.104,148.989
C09864=1133.288,144.321,-58.957,-178.844,7.106,148.988
C09865=1133.284,144.570,-58.977,-178.841,7.108,148.988
C09866=1133.279,144.820,-58.999,-178.838,7.111,148.988
C09867=1133.275,145.069,-59.019,-178.835,7.112,148.987
C09868=1133.270,145.318,-59.040,-178.833,7.114,148.987
C09869=1133.265,145.566,-59.061,-178.829,7.116,148.987
C09870=1133.260,145.816,-59.082,-178.827,7.118,148.986
C09871=1133.256,146.064,-59.102,-178.824,7.120,148.986
C09872=1133.251,146.314,-59.123,-178.821,7.123,148.986
C09873=1133.245,146.563,-59.144,-178.818,7.124,148.985
C09874=1133.241,146.811,-59.166,-178.816,7.126,148.985
C09875=1133.237,147.061,-59.187,-178.812,7.129,148.984
C09876=1133.232,147.310,-59.207,-178.810,7.130,148.984
C09877=1133.227,147.560,-59.228,-178.807,7.132,148.984
C09878=1133.222,147.808,-59.250,-178.804,7.135,148.984
C09879=1133.218,148.057,-59.270,-178.801,7.137,148.983
C09880=1133.213,148.306,-59.291,-178.799,7.138,148.983
C09881=1133.208,148.555,-59.313,-178.795,7.141,148.982
C09882=1133.204,148.805,-59.334,-178.793,7.142,148.982
C09883=1133.199,149.054,-59.355,-178.790,7.145,148.982
C09884=1133.194,149.303,-59.376,-178.787,7.147,148.981
C09885=1133.189,149.552,-59.397,-178.784,7.149,148.981
C09886=1133.184,149.801,-59.418,-178.782,7.150,148.981
C09887=1133.180,150.050,-59.440,-178.778,7.153,148.980
C09888=1133.176,150.299,-59.460,-178.776,7.155,148.980
C09889=1133.171,150.548,-59.482,-178.773,7.157,148.980
C09890=1133.166,150.797,-59.503,-178.770,7.159,148.979
C09891=1133.160,151.046,-59.524,-178.767,7.161,148.979
C09892=1133.157,151.295,-59.545,-178.765,7.163,148.979
C09893=1133.152,151.545,-59.566,-178.762,7.165,148.978
C09894=1133.147,151.793,-59.588,-178.759,7.167,148.978
C09895=1133.142,152.042,-59.609,-178.756,7.170,148.978
C09896=1133.138,152.291,-59.630,-178.753,7.171,148.977
C09897=1133.133,152.541,-59.651,-178.751,7.173,148.977
C09898=1133.128,152.789,-59.673,-178.747,7.176,148.977
C09899=1133.123,153.039,-59.694,-178.745,7.178,148.976
C09900=1133.119,153.288,-59.716,-178.742,7.179,148.976
C09901=1133.114,153.537,-59.736,-178.739,7.182,148.976
C09902=1133.109,153.786,-59.758,-178.736,7.184,148.976
C09903=1133.104,154.034,-59.780,-178.733,7.186,148.975
C09904=1133.100,154.284,-59.801,-178.730,7.188,148.975
C09905=1133.095,154.533,-59.823,-178.728,7.190,148.974
C09906=1133.090,154.782,-59.844,-178.725,7.193,148.974
C09907=1133.086,155.030,-59.865,-178.722,7.194,148.974
C09908=1133.081,155.280,-59.887,-178.719,7.197,148.973
C09909=1133.076,155.529,-59.908,-178.716,7.199,148.973
C09910=1133.071,155.778,-59.929,-178.714,7.201,148.973
C09911=1133.067,156.027,-59.951,-178.711,7.203,148.973
C09912=1133.062,156.276,-59.972,-178.708,7.205,148.972
C09913=1133.057,156.525,-59.994,-178.705,7.207,148.972
C09914=1133.053,156.774,-60.016,-178.702,7.209,148.972
C09915=1133.048,157.043,-60.039,-178.699,7.212,148.971
C09916=1133.043,157.312,-60.063,-178.696,7.214,148.971
C09917=1133.038,157.581,-60.086,-178.693,7.216,148.971
C09918=1133.033,157.850,-60.109,-178.690,7.219,148.970
C09919=1133.028,158.099,-60.131,-178.687,7.220,148.970
C09920=1133.023,158.348,-60.152,-178.684,7.223,148.970
C09921=1133.019,158.597,-60.174,-178.681,7.225,148.969
C09922=1133.013,158.846,-60.195,-178.679,7.227,148.969
C09923=1133.007,159.185,-60.225,-178.675,7.230,148.969
C09924=1132.983,160.445,-60.333,-179.484,8.827,149.569
C09925=1132.979,160.694,-60.356,-179.481,8.831,149.569
C09926=1132.975,160.943,-60.378,-179.479,8.834,149.569
C09927=1132.969,161.192,-60.400,-179.476,8.837,149.569
C09928=1132.965,161.441,-60.422,-179.474,8.840,149.569
C09929=1132.960,161.689,-60.444,-179.470,8.844,149.569
C09930=1132.956,161.939,-60.467,-179.468,8.847,149.569
C09931=1132.951,162.187,-60.489,-179.466,8.851,149.570
C09932=1132.946,162.437,-60.511,-179.463,8.854,149.570
C09933=1132.942,162.686,-60.534,-179.461,8.857,149.570
C09934=1132.937,162.934,-60.555,-179.458,8.860,149.570
C09935=1132.932,163.184,-60.578,-179.456,8.864,149.570
C09936=1132.928,163.432,-60.600,-179.453,8.868,149.570
C09937=1132.924,163.681,-60.622,-179.451,8.871,149.570
C09938=1132.919,163.931,-60.645,-179.448,8.874,149.570
C09939=1132.914,164.179,-60.667,-179.445,8.877,149.570
C09940=1132.910,164.428,-60.689,-179.443,8.880,149.570
C09941=1132.905,164.677,-60.713,-179.441,8.884,149.570
C09942=1132.900,164.926,-60.735,-179.438,8.887,149.570
C09943=1132.895,165.176,-60.757,-179.436,8.890,149.570
C09944=1132.891,165.424,-60.780,-179.433,8.893,149.570
C09945=1132.886,165.673,-60.802,-179.431,8.896,149.571
C09946=1132.882,165.922,-60.825,-179.429,8.899,149.571
C09947=1132.877,166.171,-60.847,-179.426,8.903,149.571
C09948=1132.872,166.420,-60.870,-179.424,8.906,149.571
C09949=1132.868,166.669,-60.892,-179.421,8.910,149.571
C09950=1132.863,166.917,-60.914,-179.419,8.912,149.571
C09951=1132.858,167.167,-60.937,-179.417,8.915,149.571
C09952=1132.854,167.415,-60.960,-179.414,8.918,149.571
C09953=1132.849,167.665,-60.983,-179.411,8.922,149.571
C09954=1132.845,167.913,-61.005,-179.409,8.925,149.571
C09955=1132.840,168.162,-61.028,-179.407,8.928,149.571
C09956=1132.836,168.411,-61.050,-179.404,8.931,149.571
C09957=1132.830,168.660,-61.073,-179.402,8.934,149.571
C09958=1132.826,168.909,-61.095,-179.399,8.937,149.571
C09959=1132.821,169.158,-61.119,-179.397,8.941,149.572
C09960=1132.818,169.407,-61.141,-179.395,8.944,149.572
C09961=1132.812,169.656,-61.164,-179.392,8.947,149.572
C09962=1132.807,169.905,-61.187,-179.390,8.950,149.572
C09963=1132.803,170.154,-61.210,-179.388,8.954,149.572
C09964=1132.798,170.403,-61.233,-179.386,8.956,149.572
C09965=1132.794,170.651,-61.255,-179.383,8.959,149.572
C09966=1132.789,170.900,-61.278,-179.381,8.962,149.572
C09967=1132.785,171.150,-61.300,-179.378,8.966,149.572
C09968=1132.779,171.445,-61.328,-179.376,8.969,149.572
C09969=1132.773,171.741,-61.356,-179.373,8.973,149.572
C09970=1132.769,172.037,-61.382,-179.370,8.977,149.572
C09971=1132.763,172.333,-61.410,-179.368,8.980,149.573
C09972=1132.758,172.582,-61.433,-179.365,8.983,149.573
C09973=1132.754,172.831,-61.455,-179.362,8.986,149.573
C09974=1132.749,173.080,-61.478,-179.361,8.989,149.573
C09975=1132.744,173.328,-61.501,-179.359,8.992,149.573
C09976=1132.740,173.577,-61.524,-179.356,8.995,149.573
C09977=1132.735,173.826,-61.548,-179.353,8.998,149.573
C09978=1132.730,174.075,-61.571,-179.352,9.001,149.573
C09979=1132.726,174.324,-61.594,-179.349,9.004,149.573
C09980=1132.722,174.573,-61.617,-179.347,9.007,149.573
C09981=1132.716,174.822,-61.639,-179.345,9.010,149.573
C09982=1132.711,175.071,-61.663,-179.343,9.013,149.574
C09983=1132.707,175.320,-61.685,-179.340,9.016,149.574
C09984=1132.703,175.569,-61.709,-179.338,9.019,149.574
C09985=1132.698,175.818,-61.732,-179.336,9.022,149.574
C09986=1132.693,176.067,-61.756,-179.334,9.025,149.574
C09987=1132.689,176.316,-61.778,-179.331,9.028,149.574
C09988=1132.684,176.564,-61.801,-179.330,9.031,149.574
C09989=1132.679,176.813,-61.825,-179.327,9.034,149.574
C09990=1132.675,177.062,-61.848,-179.326,9.036,149.574
C09991=1132.671,177.311,-61.871,-179.323,9.040,149.575
C09992=1132.666,177.560,-61.894,-179.321,9.043,149.575
C09993=1132.661,177.809,-61.918,-179.319,9.045,149.575
C09994=1132.656,178.058,-61.941,-179.317,9.049,149.575
C09995=1132.652,178.307,-61.964,-179.315,9.051,149.575
C09996=1132.648,178.555,-61.988,-179.312,9.054,149.575
//INST
///DATE 2021/06/25 14:32
///ATTR SC,RW,RJ
////FRAME ROBOT
///GROUP1 RB1
NOP
MOVL C00000 V=800.0 PL=0
MOVL C00001 V=800.0 PL=0
MOVL C00002 V=800.0 PL=0
MOVL C00003 V=800.0 PL=0
MOVL C00004 V=800.0 PL=0
MOVL C00005 V=800.0 PL=0
MOVL C00006 V=800.0 PL=0
MOVL C00007 V=800.0 PL=0
MOVL C00008 V=800.0 PL=0
MOVL C00009 V=800.0 PL=0
MOVL C00010 V=800.0 PL=0
MOVL C00011 V=800.0 PL=0
MOVL C00012 V=800.0 PL=0
MOVL C00013 V=800.0 PL=0
MOVL C00014 V=800.0 PL=0
MOVL C00015 V=800.0 PL=0
MOVL C00016 V=800.0 PL=0
MOVL C00017 V=800.0 PL=0
MOVL C00018 V=800.0 PL=0
MOVL C00019 V=800.0 PL=0
MOVL C00020 V=800.0 PL=0
MOVL C00021 V=800.0 PL=0
MOVL C00022 V=800.0 PL=0
MOVL C00023 V=800.0 PL=0
MOVL C00024 V=800.0 PL=0
MOVL C00025 V=800.0 PL=0
MOVL C00026 V=800.0 PL=0
MOVL C00027 V=800.0 PL=0
MOVL C00028 V=800.0 PL=0
MOVL C00029 V=800.0 PL=0
MOVL C00030 V=800.0 PL=0
MOVL C00031 V=800.0 PL=0
MOVL C00032 V=800.0 PL=0
MOVL C00033 V=800.0 PL=0
MOVL C00034 V=800.0 PL=0
MOVL C00035 V=800.0 PL=0
MOVL C00036 V=800.0 PL=0
MOVL C00037 V=800.0 PL=0
MOVL C00038 V=800.0 PL=0
MOVL C00039 V=800.0 PL=0
MOVL C00040 V=800.0 PL=0
MOVL C00041 V=800.0 PL=0
MOVL C00042 V=800.0 PL=0
MOVL C00043 V=800.0 PL=0
MOVL C00044 V=800.0 PL=0
MOVL C00045 V=800.0 PL=0
MOVL C00046 V=800.0 PL=0
MOVL C00047 V=800.0 PL=0
MOVL C00048 V=800.0 PL=0
MOVL C00049 V=800.0 PL=0
MOVL C00050 V=800.0 PL=0
MOVL C00051 V=800.0 PL=0
MOVL C00052 V=800.0 PL=0
MOVL C00053 V=800.0 PL=0
MOVL C00054 V=800.0 PL=0
MOVL C00055 V=800.0 PL=0
MOVL C00056 V=800.0 PL=0
MOVL C00057 V=800.0 PL=0
MOVL C00058 V=800.0 PL=0
MOVL C00059 V=800.0 PL=0
MOVL C00060 V=800.0 PL=0
MOVL C00061 V=800.0 PL=0
MOVL C00062 V=800.0 PL=0
MOVL C00063 V=800.0 PL=0
MOVL C00064 V=800.0 PL=0
MOVL C00065 V=800.0 PL=0
MOVL C00066 V=800.0 PL=0
MOVL C00067 V=800.0 PL=0
MOVL C00068 V=800.0 PL=0
MOVL C00069 V=800.0 PL=0
MOVL C00070 V=800.0 PL=0
MOVL C00071 V=800.0 PL=0
MOVL C00072 V=800.0 PL=0
MOVL C00073 V=800.0 PL=0
MOVL C00074 V=800.0 PL=0
MOVL C00075 V=800.0 PL=0
MOVL C00076 V=800.0 PL=0
MOVL C00077 V=800.0 PL=0
MOVL C00078 V=800.0 PL=0
MOVL C00079 V=800.0 PL=0
MOVL C00080 V=800.0 PL=0
MOVL C00081 V=800.0 PL=0
MOVL C00082 V=800.0 PL=0
MOVL C00083 V=800.0 PL=0
MOVL C00084 V=800.0 PL=0
MOVL C00085 V=800.0 PL=0
MOVL C00086 V=800.0 PL=0
MOVL C00087 V=800.0 PL=0
MOVL C00088 V=800.0 PL=0
MOVL C00089 V=800.0 PL=0
MOVL C00090 V=800.0 PL=0
MOVL C00091 V=800.0 PL=0
MOVL C00092 V=800.0 PL=0
MOVL C00093 V=800.0 PL=0
MOVL C00094 V=800.0 PL=0
MOVL C00095 V=800.0 PL=0
MOVL C00096 V=800.0 PL=0
MOVL C00097 V=800.0 PL=0
MOVL C00098 V=800.0 PL=0
MOVL C00099 V=800.0 PL=0
MOVL C00100 V=800.0 PL=0
MOVL C00101 V=800.0 PL=0
MOVL C00102 V=800.0 PL=0
MOVL C00103 V=800.0 PL=0
MOVL C00104 V=800.0 PL=0
MOVL C00105 V=800.0 PL=0
MOVL C00106 V=800.0 PL=0
MOVL C00107 V=800.0 PL=0
MOVL C00108 V=800.0 PL=0
MOVL C00109 V=800.0 PL=0
MOVL C00110 V=800.0 PL=0
MOVL C00111 V=800.0 PL=0
MOVL C00112 V=800.0 PL=0
MOVL C00113 V=800.0 PL=0
MOVL C00114 V=800.0 PL=0
MOVL C00115 V=800.0 PL=0
MOVL C00116 V=800.0 PL=0
MOVL C00117 V=800.0 PL=0
MOVL C00118 V=800.0 PL=0
MOVL C00119 V=800.0 PL=0
MOVL C00120 V=800.0 PL=0
MOVL C00121 V=800.0 PL=0
MOVL C00122 V=800.0 PL=0
MOVL C00123 V=800.0 PL=0
MOVL C00124 V=800.0 PL=0
MOVL C00125 V=800.0 PL=0
MOVL C00126 V=800.0 PL=0
MOVL C00127 V=800.0 PL=0
MOVL C00128 V=800.0 PL=0
MOVL C00129 V=800.0 PL=0
MOVL C00130 V=800.0 PL=0
MOVL C00131 V=800.0 PL=0
MOVL C00132 V=800.0 PL=0
MOVL C00133 V=800.0 PL=0
MOVL C00134 V=800.0 PL=0
MOVL C00135 V=800.0 PL=0
MOVL C00136 V=800.0 PL=0
MOVL C00137 V=800.0 PL=0
MOVL C00138 V=800.0 PL=0
MOVL C00139 V=800.0 PL=0
MOVL C00140 V=800.0 PL=0
MOVL C00141 V=800.0 PL=0
MOVL C00142 V=800.0 PL=0
MOVL C00143 V=800.0 PL=0
MOVL C00144 V=800.0 PL=0
MOVL C00145 V=800.0 PL=0
MOVL C00146 V=800.0 PL=0
MOVL C00147 V=800.0 PL=0
MOVL C00148 V=800.0 PL=0
MOVL C00149 V=800.0 PL=0
MOVL C00150 V=800.0 PL=0
MOVL C00151 V=800.0 PL=0
MOVL C00152 V=800.0 PL=0
MOVL C00153 V=800.0 PL=0
MOVL C00154 V=800.0 PL=0
MOVL C00155 V=800.0 PL=0
MOVL C00156 V=800.0 PL=0
MOVL C00157 V=800.0 PL=0
MOVL C00158 V=800.0 PL=0
MOVL C00159 V=800.0 PL=0
MOVL C00160 V=800.0 PL=0
MOVL C00161 V=800.0 PL=0
MOVL C00162 V=800.0 PL=0
MOVL C00163 V=800.0 PL=0
MOVL C00164 V=800.0 PL=0
MOVL C00165 V=800.0 PL=0
MOVL C00166 V=800.0 PL=0
MOVL C00167 V=800.0 PL=0
MOVL C00168 V=800.0 PL=0
MOVL C00169 V=800.0 PL=0
MOVL C00170 V=800.0 PL=0
MOVL C00171 V=800.0 PL=0
MOVL C00172 V=800.0 PL=0
MOVL C00173 V=800.0 PL=0
MOVL C00174 V=800.0 PL=0
MOVL C00175 V=800.0 PL=0
MOVL C00176 V=800.0 PL=0
MOVL C00177 V=800.0 PL=0
MOVL C00178 V=800.0 PL=0
MOVL C00179 V=800.0 PL=0
MOVL C00180 V=800.0 PL=0
MOVL C00181 V=800.0 PL=0
MOVL C00182 V=800.0 PL=0
MOVL C00183 V=800.0 PL=0
MOVL C00184 V=800.0 PL=0
MOVL C00185 V=800.0 PL=0
MOVL C00186 V=800.0 PL=0
MOVL C00187 V=800.0 PL=0
MOVL C00188 V=800.0 PL=0
MOVL C00189 V=800.0 PL=0
MOVL C00190 V=800.0 PL=0
MOVL C00191 V=800.0 PL=0
MOVL C00192 V=800.0 PL=0
MOVL C00193 V=800.0 PL=0
MOVL C00194 V=800.0 PL=0
MOVL C00195 V=800.0 PL=0
MOVL C00196 V=800.0 PL=0
MOVL C00197 V=800.0 PL=0
MOVL C00198 V=800.0 PL=0
MOVL C00199 V=800.0 PL=0
MOVL C00200 V=800.0 PL=0
MOVL C00201 V=800.0 PL=0
MOVL C00202 V=800.0 PL=0
MOVL C00203 V=800.0 PL=0
MOVL C00204 V=800.0 PL=0
MOVL C00205 V=800.0 PL=0
MOVL C00206 V=800.0 PL=0
MOVL C00207 V=800.0 PL=0
MOVL C00208 V=800.0 PL=0
MOVL C00209 V=800.0 PL=0
MOVL C00210 V=800.0 PL=0
MOVL C00211 V=800.0 PL=0
MOVL C00212 V=800.0 PL=0
MOVL C00213 V=800.0 PL=0
MOVL C00214 V=800.0 PL=0
MOVL C00215 V=800.0 PL=0
MOVL C00216 V=800.0 PL=0
MOVL C00217 V=800.0 PL=0
MOVL C00218 V=800.0 PL=0
MOVL C00219 V=800.0 PL=0
MOVL C00220 V=800.0 PL=0
MOVL C00221 V=800.0 PL=0
MOVL C00222 V=800.0 PL=0
MOVL C00223 V=800.0 PL=0
MOVL C00224 V=800.0 PL=0
MOVL C00225 V=800.0 PL=0
MOVL C00226 V=800.0 PL=0
MOVL C00227 V=800.0 PL=0
MOVL C00228 V=800.0 PL=0
MOVL C00229 V=800.0 PL=0
MOVL C00230 V=800.0 PL=0
MOVL C00231 V=800.0 PL=0
MOVL C00232 V=800.0 PL=0
MOVL C00233 V=800.0 PL=0
MOVL C00234 V=800.0 PL=0
MOVL C00235 V=800.0 PL=0
MOVL C00236 V=800.0 PL=0
MOVL C00237 V=800.0 PL=0
MOVL C00238 V=800.0 PL=0
MOVL C00239 V=800.0 PL=0
MOVL C00240 V=800.0 PL=0
MOVL C00241 V=800.0 PL=0
MOVL C00242 V=800.0 PL=0
MOVL C00243 V=800.0 PL=0
MOVL C00244 V=800.0 PL=0
MOVL C00245 V=800.0 PL=0
MOVL C00246 V=800.0 PL=0
MOVL C00247 V=800.0 PL=0
MOVL C00248 V=800.0 PL=0
MOVL C00249 V=800.0 PL=0
MOVL C00250 V=800.0 PL=0
MOVL C00251 V=800.0 PL=0
MOVL C00252 V=800.0 PL=0
MOVL C00253 V=800.0 PL=0
MOVL C00254 V=800.0 PL=0
MOVL C00255 V=800.0 PL=0
MOVL C00256 V=800.0 PL=0
MOVL C00257 V=800.0 PL=0
MOVL C00258 V=800.0 PL=0
MOVL C00259 V=800.0 PL=0
MOVL C00260 V=800.0 PL=0
MOVL C00261 V=800.0 PL=0
MOVL C00262 V=800.0 PL=0
MOVL C00263 V=800.0 PL=0
MOVL C00264 V=800.0 PL=0
MOVL C00265 V=800.0 PL=0
MOVL C00266 V=800.0 PL=0
MOVL C00267 V=800.0 PL=0
MOVL C00268 V=800.0 PL=0
MOVL C00269 V=800.0 PL=0
MOVL C00270 V=800.0 PL=0
MOVL C00271 V=800.0 PL=0
MOVL C00272 V=800.0 PL=0
MOVL C00273 V=800.0 PL=0
MOVL C00274 V=800.0 PL=0
MOVL C00275 V=800.0 PL=0
MOVL C00276 V=800.0 PL=0
MOVL C00277 V=800.0 PL=0
MOVL C00278 V=800.0 PL=0
MOVL C00279 V=800.0 PL=0
MOVL C00280 V=800.0 PL=0
MOVL C00281 V=800.0 PL=0
MOVL C00282 V=800.0 PL=0
MOVL C00283 V=800.0 PL=0
MOVL C00284 V=800.0 PL=0
MOVL C00285 V=800.0 PL=0
MOVL C00286 V=800.0 PL=0
MOVL C00287 V=800.0 PL=0
MOVL C00288 V=800.0 PL=0
MOVL C00289 V=800.0 PL=0
MOVL C00290 V=800.0 PL=0
MOVL C00291 V=800.0 PL=0
MOVL C00292 V=800.0 PL=0
MOVL C00293 V=800.0 PL=0
MOVL C00294 V=800.0 PL=0
MOVL C00295 V=800.0 PL=0
MOVL C00296 V=800.0 PL=0
MOVL C00297 V=800.0 PL=0
MOVL C00298 V=800.0 PL=0
MOVL C00299 V=800.0 PL=0
MOVL C00300 V=800.0 PL=0
MOVL C00301 V=800.0 PL=0
MOVL C00302 V=800.0 PL=0
MOVL C00303 V=800.0 PL=0
MOVL C00304 V=800.0 PL=0
MOVL C00305 V=800.0 PL=0
MOVL C00306 V=800.0 PL=0
MOVL C00307 V=800.0 PL=0
MOVL C00308 V=800.0 PL=0
MOVL C00309 V=800.0 PL=0
MOVL C00310 V=800.0 PL=0
MOVL C00311 V=800.0 PL=0
MOVL C00312 V=800.0 PL=0
MOVL C00313 V=800.0 PL=0
MOVL C00314 V=800.0 PL=0
MOVL C00315 V=800.0 PL=0
MOVL C00316 V=800.0 PL=0
MOVL C00317 V=800.0 PL=0
MOVL C00318 V=800.0 PL=0
MOVL C00319 V=800.0 PL=0
MOVL C00320 V=800.0 PL=0
MOVL C00321 V=800.0 PL=0
MOVL C00322 V=800.0 PL=0
MOVL C00323 V=800.0 PL=0
MOVL C00324 V=800.0 PL=0
MOVL C00325 V=800.0 PL=0
MOVL C00326 V=800.0 PL=0
MOVL C00327 V=800.0 PL=0
MOVL C00328 V=800.0 PL=0
MOVL C00329 V=800.0 PL=0
MOVL C00330 V=800.0 PL=0
MOVL C00331 V=800.0 PL=0
MOVL C00332 V=800.0 PL=0
MOVL C00333 V=800.0 PL=0
MOVL C00334 V=800.0 PL=0
MOVL C00335 V=800.0 PL=0
MOVL C00336 V=800.0 PL=0
MOVL C00337 V=800.0 PL=0
MOVL C00338 V=800.0 PL=0
MOVL C00339 V=800.0 PL=0
MOVL C00340 V=800.0 PL=0
MOVL C00341 V=800.0 PL=0
MOVL C00342 V=800.0 PL=0
MOVL C00343 V=800.0 PL=0
MOVL C00344 V=800.0 PL=0
MOVL C00345 V=800.0 PL=0
MOVL C00346 V=800.0 PL=0
MOVL C00347 V=800.0 PL=0
MOVL C00348 V=800.0 PL=0
MOVL C00349 V=800.0 PL=0
MOVL C00350 V=800.0 PL=0
MOVL C00351 V=800.0 PL=0
MOVL C00352 V=800.0 PL=0
MOVL C00353 V=800.0 PL=0
MOVL C00354 V=800.0 PL=0
MOVL C00355 V=800.0 PL=0
MOVL C00356 V=800.0 PL=0
MOVL C00357 V=800.0 PL=0
MOVL C00358 V=800.0 PL=0
MOVL C00359 V=800.0 PL=0
MOVL C00360 V=800.0 PL=0
MOVL C00361 V=800.0 PL=0
MOVL C00362 V=800.0 PL=0
MOVL C00363 V=800.0 PL=0
MOVL C00364 V=800.0 PL=0
MOVL C00365 V=800.0 PL=0
MOVL C00366 V=800.0 PL=0
MOVL C00367 V=800.0 PL=0
MOVL C00368 V=800.0 PL=0
MOVL C00369 V=800.0 PL=0
MOVL C00370 V=800.0 PL=0
MOVL C00371 V=800.0 PL=0
MOVL C00372 V=800.0 PL=0
MOVL C00373 V=800.0 PL=0
MOVL C00374 V=800.0 PL=0
MOVL C00375 V=800.0 PL=0
MOVL C00376 V=800.0 PL=0
MOVL C00377 V=800.0 PL=0
MOVL C00378 V=800.0 PL=0
MOVL C00379 V=800.0 PL=0
MOVL C00380 V=800.0 PL=0
MOVL C00381 V=800.0 PL=0
MOVL C00382 V=800.0 PL=0
MOVL C00383 V=800.0 PL=0
MOVL C00384 V=800.0 PL=0
MOVL C00385 V=800.0 PL=0
MOVL C00386 V=800.0 PL=0
MOVL C00387 V=800.0 PL=0
MOVL C00388 V=800.0 PL=0
MOVL C00389 V=800.0 PL=0
MOVL C00390 V=800.0 PL=0
MOVL C00391 V=800.0 PL=0
MOVL C00392 V=800.0 PL=0
MOVL C00393 V=800.0 PL=0
MOVL C00394 V=800.0 PL=0
MOVL C00395 V=800.0 PL=0
MOVL C00396 V=800.0 PL=0
MOVL C00397 V=800.0 PL=0
MOVL C00398 V=800.0 PL=0
MOVL C00399 V=800.0 PL=0
MOVL C00400 V=800.0 PL=0
MOVL C00401 V=800.0 PL=0
MOVL C00402 V=800.0 PL=0
MOVL C00403 V=800.0 PL=0
MOVL C00404 V=800.0 PL=0
MOVL C00405 V=800.0 PL=0
MOVL C00406 V=800.0 PL=0
MOVL C00407 V=800.0 PL=0
MOVL C00408 V=800.0 PL=0
MOVL C00409 V=800.0 PL=0
MOVL C00410 V=800.0 PL=0
MOVL C00411 V=800.0 PL=0
MOVL C00412 V=800.0 PL=0
MOVL C00413 V=800.0 PL=0
MOVL C00414 V=800.0 PL=0
MOVL C00415 V=800.0 PL=0
MOVL C00416 V=800.0 PL=0
MOVL C00417 V=800.0 PL=0
MOVL C00418 V=800.0 PL=0
MOVL C00419 V=800.0 PL=0
MOVL C00420 V=800.0 PL=0
MOVL C00421 V=800.0 PL=0
MOVL C00422 V=800.0 PL=0
MOVL C00423 V=800.0 PL=0
MOVL C00424 V=800.0 PL=0
MOVL C00425 V=800.0 PL=0
MOVL C00426 V=800.0 PL=0
MOVL C00427 V=800.0 PL=0
MOVL C00428 V=800.0 PL=0
MOVL C00429 V=800.0 PL=0
MOVL C00430 V=800.0 PL=0
MOVL C00431 V=800.0 PL=0
MOVL C00432 V=800.0 PL=0
MOVL C00433 V=800.0 PL=0
MOVL C00434 V=800.0 PL=0
MOVL C00435 V=800.0 PL=0
MOVL C00436 V=800.0 PL=0
MOVL C00437 V=800.0 PL=0
MOVL C00438 V=800.0 PL=0
MOVL C00439 V=800.0 PL=0
MOVL C00440 V=800.0 PL=0
MOVL C00441 V=800.0 PL=0
MOVL C00442 V=800.0 PL=0
MOVL C00443 V=800.0 PL=0
MOVL C00444 V=800.0 PL=0
MOVL C00445 V=800.0 PL=0
MOVL C00446 V=800.0 PL=0
MOVL C00447 V=800.0 PL=0
MOVL C00448 V=800.0 PL=0
MOVL C00449 V=800.0 PL=0
MOVL C00450 V=800.0 PL=0
MOVL C00451 V=800.0 PL=0
MOVL C00452 V=800.0 PL=0
MOVL C00453 V=800.0 PL=0
MOVL C00454 V=800.0 PL=0
MOVL C00455 V=800.0 PL=0
MOVL C00456 V=800.0 PL=0
MOVL C00457 V=800.0 PL=0
MOVL C00458 V=800.0 PL=0
MOVL C00459 V=800.0 PL=0
MOVL C00460 V=800.0 PL=0
MOVL C00461 V=800.0 PL=0
MOVL C00462 V=800.0 PL=0
MOVL C00463 V=800.0 PL=0
MOVL C00464 V=800.0 PL=0
MOVL C00465 V=800.0 PL=0
MOVL C00466 V=800.0 PL=0
MOVL C00467 V=800.0 PL=0
MOVL C00468 V=800.0 PL=0
MOVL C00469 V=800.0 PL=0
MOVL C00470 V=800.0 PL=0
MOVL C00471 V=800.0 PL=0
MOVL C00472 V=800.0 PL=0
MOVL C00473 V=800.0 PL=0
MOVL C00474 V=800.0 PL=0
MOVL C00475 V=800.0 PL=0
MOVL C00476 V=800.0 PL=0
MOVL C00477 V=800.0 PL=0
MOVL C00478 V=800.0 PL=0
MOVL C00479 V=800.0 PL=0
MOVL C00480 V=800.0 PL=0
MOVL C00481 V=800.0 PL=0
MOVL C00482 V=800.0 PL=0
MOVL C00483 V=800.0 PL=0
MOVL C00484 V=800.0 PL=0
MOVL C00485 V=800.0 PL=0
MOVL C00486 V=800.0 PL=0
MOVL C00487 V=800.0 PL=0
MOVL C00488 V=800.0 PL=0
MOVL C00489 V=800.0 PL=0
MOVL C00490 V=800.0 PL=0
MOVL C00491 V=800.0 PL=0
MOVL C00492 V=800.0 PL=0
MOVL C00493 V=800.0 PL=0
MOVL C00494 V=800.0 PL=0
MOVL C00495 V=800.0 PL=0
MOVL C00496 V=800.0 PL=0
MOVL C00497 V=800.0 PL=0
MOVL C00498 V=800.0 PL=0
MOVL C00499 V=800.0 PL=0
MOVL C00500 V=800.0 PL=0
MOVL C00501 V=800.0 PL=0
MOVL C00502 V=800.0 PL=0
MOVL C00503 V=800.0 PL=0
MOVL C00504 V=800.0 PL=0
MOVL C00505 V=800.0 PL=0
MOVL C00506 V=800.0 PL=0
MOVL C00507 V=800.0 PL=0
MOVL C00508 V=800.0 PL=0
MOVL C00509 V=800.0 PL=0
MOVL C00510 V=800.0 PL=0
MOVL C00511 V=800.0 PL=0
MOVL C00512 V=800.0 PL=0
MOVL C00513 V=800.0 PL=0
MOVL C00514 V=800.0 PL=0
MOVL C00515 V=800.0 PL=0
MOVL C00516 V=800.0 PL=0
MOVL C00517 V=800.0 PL=0
MOVL C00518 V=800.0 PL=0
MOVL C00519 V=800.0 PL=0
MOVL C00520 V=800.0 PL=0
MOVL C00521 V=800.0 PL=0
MOVL C00522 V=800.0 PL=0
MOVL C00523 V=800.0 PL=0
MOVL C00524 V=800.0 PL=0
MOVL C00525 V=800.0 PL=0
MOVL C00526 V=800.0 PL=0
MOVL C00527 V=800.0 PL=0
MOVL C00528 V=800.0 PL=0
MOVL C00529 V=800.0 PL=0
MOVL C00530 V=800.0 PL=0
MOVL C00531 V=800.0 PL=0
MOVL C00532 V=800.0 PL=0
MOVL C00533 V=800.0 PL=0
MOVL C00534 V=800.0 PL=0
MOVL C00535 V=800.0 PL=0
MOVL C00536 V=800.0 PL=0
MOVL C00537 V=800.0 PL=0
MOVL C00538 V=800.0 PL=0
MOVL C00539 V=800.0 PL=0
MOVL C00540 V=800.0 PL=0
MOVL C00541 V=800.0 PL=0
MOVL C00542 V=800.0 PL=0
MOVL C00543 V=800.0 PL=0
MOVL C00544 V=800.0 PL=0
MOVL C00545 V=800.0 PL=0
MOVL C00546 V=800.0 PL=0
MOVL C00547 V=800.0 PL=0
MOVL C00548 V=800.0 PL=0
MOVL C00549 V=800.0 PL=0
MOVL C00550 V=800.0 PL=0
MOVL C00551 V=800.0 PL=0
MOVL C00552 V=800.0 PL=0
MOVL C00553 V=800.0 PL=0
MOVL C00554 V=800.0 PL=0
MOVL C00555 V=800.0 PL=0
MOVL C00556 V=800.0 PL=0
MOVL C00557 V=800.0 PL=0
MOVL C00558 V=800.0 PL=0
MOVL C00559 V=800.0 PL=0
MOVL C00560 V=800.0 PL=0
MOVL C00561 V=800.0 PL=0
MOVL C00562 V=800.0 PL=0
MOVL C00563 V=800.0 PL=0
MOVL C00564 V=800.0 PL=0
MOVL C00565 V=800.0 PL=0
MOVL C00566 V=800.0 PL=0
MOVL C00567 V=800.0 PL=0
MOVL C00568 V=800.0 PL=0
MOVL C00569 V=800.0 PL=0
MOVL C00570 V=800.0 PL=0
MOVL C00571 V=800.0 PL=0
MOVL C00572 V=800.0 PL=0
MOVL C00573 V=800.0 PL=0
MOVL C00574 V=800.0 PL=0
MOVL C00575 V=800.0 PL=0
MOVL C00576 V=800.0 PL=0
MOVL C00577 V=800.0 PL=0
MOVL C00578 V=800.0 PL=0
MOVL C00579 V=800.0 PL=0
MOVL C00580 V=800.0 PL=0
MOVL C00581 V=800.0 PL=0
MOVL C00582 V=800.0 PL=0
MOVL C00583 V=800.0 PL=0
MOVL C00584 V=800.0 PL=0
MOVL C00585 V=800.0 PL=0
MOVL C00586 V=800.0 PL=0
MOVL C00587 V=800.0 PL=0
MOVL C00588 V=800.0 PL=0
MOVL C00589 V=800.0 PL=0
MOVL C00590 V=800.0 PL=0
MOVL C00591 V=800.0 PL=0
MOVL C00592 V=800.0 PL=0
MOVL C00593 V=800.0 PL=0
MOVL C00594 V=800.0 PL=0
MOVL C00595 V=800.0 PL=0
MOVL C00596 V=800.0 PL=0
MOVL C00597 V=800.0 PL=0
MOVL C00598 V=800.0 PL=0
MOVL C00599 V=800.0 PL=0
MOVL C00600 V=800.0 PL=0
MOVL C00601 V=800.0 PL=0
MOVL C00602 V=800.0 PL=0
MOVL C00603 V=800.0 PL=0
MOVL C00604 V=800.0 PL=0
MOVL C00605 V=800.0 PL=0
MOVL C00606 V=800.0 PL=0
MOVL C00607 V=800.0 PL=0
MOVL C00608 V=800.0 PL=0
MOVL C00609 V=800.0 PL=0
MOVL C00610 V=800.0 PL=0
MOVL C00611 V=800.0 PL=0
MOVL C00612 V=800.0 PL=0
MOVL C00613 V=800.0 PL=0
MOVL C00614 V=800.0 PL=0
MOVL C00615 V=800.0 PL=0
MOVL C00616 V=800.0 PL=0
MOVL C00617 V=800.0 PL=0
MOVL C00618 V=800.0 PL=0
MOVL C00619 V=800.0 PL=0
MOVL C00620 V=800.0 PL=0
MOVL C00621 V=800.0 PL=0
MOVL C00622 V=800.0 PL=0
MOVL C00623 V=800.0 PL=0
MOVL C00624 V=800.0 PL=0
MOVL C00625 V=800.0 PL=0
MOVL C00626 V=800.0 PL=0
MOVL C00627 V=800.0 PL=0
MOVL C00628 V=800.0 PL=0
MOVL C00629 V=800.0 PL=0
MOVL C00630 V=800.0 PL=0
MOVL C00631 V=800.0 PL=0
MOVL C00632 V=800.0 PL=0
MOVL C00633 V=800.0 PL=0
MOVL C00634 V=800.0 PL=0
MOVL C00635 V=800.0 PL=0
MOVL C00636 V=800.0 PL=0
MOVL C00637 V=800.0 PL=0
MOVL C00638 V=800.0 PL=0
MOVL C00639 V=800.0 PL=0
MOVL C00640 V=800.0 PL=0
MOVL C00641 V=800.0 PL=0
MOVL C00642 V=800.0 PL=0
MOVL C00643 V=800.0 PL=0
MOVL C00644 V=800.0 PL=0
MOVL C00645 V=800.0 PL=0
MOVL C00646 V=800.0 PL=0
MOVL C00647 V=800.0 PL=0
MOVL C00648 V=800.0 PL=0
MOVL C00649 V=800.0 PL=0
MOVL C00650 V=800.0 PL=0
MOVL C00651 V=800.0 PL=0
MOVL C00652 V=800.0 PL=0
MOVL C00653 V=800.0 PL=0
MOVL C00654 V=800.0 PL=0
MOVL C00655 V=800.0 PL=0
MOVL C00656 V=800.0 PL=0
MOVL C00657 V=800.0 PL=0
MOVL C00658 V=800.0 PL=0
MOVL C00659 V=800.0 PL=0
MOVL C00660 V=800.0 PL=0
MOVL C00661 V=800.0 PL=0
MOVL C00662 V=800.0 PL=0
MOVL C00663 V=800.0 PL=0
MOVL C00664 V=800.0 PL=0
MOVL C00665 V=800.0 PL=0
MOVL C00666 V=800.0 PL=0
MOVL C00667 V=800.0 PL=0
MOVL C00668 V=800.0 PL=0
MOVL C00669 V=800.0 PL=0
MOVL C00670 V=800.0 PL=0
MOVL C00671 V=800.0 PL=0
MOVL C00672 V=800.0 PL=0
MOVL C00673 V=800.0 PL=0
MOVL C00674 V=800.0 PL=0
MOVL C00675 V=800.0 PL=0
MOVL C00676 V=800.0 PL=0
MOVL C00677 V=800.0 PL=0
MOVL C00678 V=800.0 PL=0
MOVL C00679 V=800.0 PL=0
MOVL C00680 V=800.0 PL=0
MOVL C00681 V=800.0 PL=0
MOVL C00682 V=800.0 PL=0
MOVL C00683 V=800.0 PL=0
MOVL C00684 V=800.0 PL=0
MOVL C00685 V=800.0 PL=0
MOVL C00686 V=800.0 PL=0
MOVL C00687 V=800.0 PL=0
MOVL C00688 V=800.0 PL=0
MOVL C00689 V=800.0 PL=0
MOVL C00690 V=800.0 PL=0
MOVL C00691 V=800.0 PL=0
MOVL C00692 V=800.0 PL=0
MOVL C00693 V=800.0 PL=0
MOVL C00694 V=800.0 PL=0
MOVL C00695 V=800.0 PL=0
MOVL C00696 V=800.0 PL=0
MOVL C00697 V=800.0 PL=0
MOVL C00698 V=800.0 PL=0
MOVL C00699 V=800.0 PL=0
MOVL C00700 V=800.0 PL=0
MOVL C00701 V=800.0 PL=0
MOVL C00702 V=800.0 PL=0
MOVL C00703 V=800.0 PL=0
MOVL C00704 V=800.0 PL=0
MOVL C00705 V=800.0 PL=0
MOVL C00706 V=800.0 PL=0
MOVL C00707 V=800.0 PL=0
MOVL C00708 V=800.0 PL=0
MOVL C00709 V=800.0 PL=0
MOVL C00710 V=800.0 PL=0
MOVL C00711 V=800.0 PL=0
MOVL C00712 V=800.0 PL=0
MOVL C00713 V=800.0 PL=0
MOVL C00714 V=800.0 PL=0
MOVL C00715 V=800.0 PL=0
MOVL C00716 V=800.0 PL=0
MOVL C00717 V=800.0 PL=0
MOVL C00718 V=800.0 PL=0
MOVL C00719 V=800.0 PL=0
MOVL C00720 V=800.0 PL=0
MOVL C00721 V=800.0 PL=0
MOVL C00722 V=800.0 PL=0
MOVL C00723 V=800.0 PL=0
MOVL C00724 V=800.0 PL=0
MOVL C00725 V=800.0 PL=0
MOVL C00726 V=800.0 PL=0
MOVL C00727 V=800.0 PL=0
MOVL C00728 V=800.0 PL=0
MOVL C00729 V=800.0 PL=0
MOVL C00730 V=800.0 PL=0
MOVL C00731 V=800.0 PL=0
MOVL C00732 V=800.0 PL=0
MOVL C00733 V=800.0 PL=0
MOVL C00734 V=800.0 PL=0
MOVL C00735 V=800.0 PL=0
MOVL C00736 V=800.0 PL=0
MOVL C00737 V=800.0 PL=0
MOVL C00738 V=800.0 PL=0
MOVL C00739 V=800.0 PL=0
MOVL C00740 V=800.0 PL=0
MOVL C00741 V=800.0 PL=0
MOVL C00742 V=800.0 PL=0
MOVL C00743 V=800.0 PL=0
MOVL C00744 V=800.0 PL=0
MOVL C00745 V=800.0 PL=0
MOVL C00746 V=800.0 PL=0
MOVL C00747 V=800.0 PL=0
MOVL C00748 V=800.0 PL=0
MOVL C00749 V=800.0 PL=0
MOVL C00750 V=800.0 PL=0
MOVL C00751 V=800.0 PL=0
MOVL C00752 V=800.0 PL=0
MOVL C00753 V=800.0 PL=0
MOVL C00754 V=800.0 PL=0
MOVL C00755 V=800.0 PL=0
MOVL C00756 V=800.0 PL=0
MOVL C00757 V=800.0 PL=0
MOVL C00758 V=800.0 PL=0
MOVL C00759 V=800.0 PL=0
MOVL C00760 V=800.0 PL=0
MOVL C00761 V=800.0 PL=0
MOVL C00762 V=800.0 PL=0
MOVL C00763 V=800.0 PL=0
MOVL C00764 V=800.0 PL=0
MOVL C00765 V=800.0 PL=0
MOVL C00766 V=800.0 PL=0
MOVL C00767 V=800.0 PL=0
MOVL C00768 V=800.0 PL=0
MOVL C00769 V=800.0 PL=0
MOVL C00770 V=800.0 PL=0
MOVL C00771 V=800.0 PL=0
MOVL C00772 V=800.0 PL=0
MOVL C00773 V=800.0 PL=0
MOVL C00774 V=800.0 PL=0
MOVL C00775 V=800.0 PL=0
MOVL C00776 V=800.0 PL=0
MOVL C00777 V=800.0 PL=0
MOVL C00778 V=800.0 PL=0
MOVL C00779 V=800.0 PL=0
MOVL C00780 V=800.0 PL=0
MOVL C00781 V=800.0 PL=0
MOVL C00782 V=800.0 PL=0
MOVL C00783 V=800.0 PL=0
MOVL C00784 V=800.0 PL=0
MOVL C00785 V=800.0 PL=0
MOVL C00786 V=800.0 PL=0
MOVL C00787 V=800.0 PL=0
MOVL C00788 V=800.0 PL=0
MOVL C00789 V=800.0 PL=0
MOVL C00790 V=800.0 PL=0
MOVL C00791 V=800.0 PL=0
MOVL C00792 V=800.0 PL=0
MOVL C00793 V=800.0 PL=0
MOVL C00794 V=800.0 PL=0
MOVL C00795 V=800.0 PL=0
MOVL C00796 V=800.0 PL=0
MOVL C00797 V=800.0 PL=0
MOVL C00798 V=800.0 PL=0
MOVL C00799 V=800.0 PL=0
MOVL C00800 V=800.0 PL=0
MOVL C00801 V=800.0 PL=0
MOVL C00802 V=800.0 PL=0
MOVL C00803 V=800.0 PL=0
MOVL C00804 V=800.0 PL=0
MOVL C00805 V=800.0 PL=0
MOVL C00806 V=800.0 PL=0
MOVL C00807 V=800.0 PL=0
MOVL C00808 V=800.0 PL=0
MOVL C00809 V=800.0 PL=0
MOVL C00810 V=800.0 PL=0
MOVL C00811 V=800.0 PL=0
MOVL C00812 V=800.0 PL=0
MOVL C00813 V=800.0 PL=0
MOVL C00814 V=800.0 PL=0
MOVL C00815 V=800.0 PL=0
MOVL C00816 V=800.0 PL=0
MOVL C00817 V=800.0 PL=0
MOVL C00818 V=800.0 PL=0
MOVL C00819 V=800.0 PL=0
MOVL C00820 V=800.0 PL=0
MOVL C00821 V=800.0 PL=0
MOVL C00822 V=800.0 PL=0
MOVL C00823 V=800.0 PL=0
MOVL C00824 V=800.0 PL=0
MOVL C00825 V=800.0 PL=0
MOVL C00826 V=800.0 PL=0
MOVL C00827 V=800.0 PL=0
MOVL C00828 V=800.0 PL=0
MOVL C00829 V=800.0 PL=0
MOVL C00830 V=800.0 PL=0
MOVL C00831 V=800.0 PL=0
MOVL C00832 V=800.0 PL=0
MOVL C00833 V=800.0 PL=0
MOVL C00834 V=800.0 PL=0
MOVL C00835 V=800.0 PL=0
MOVL C00836 V=800.0 PL=0
MOVL C00837 V=800.0 PL=0
MOVL C00838 V=800.0 PL=0
MOVL C00839 V=800.0 PL=0
MOVL C00840 V=800.0 PL=0
MOVL C00841 V=800.0 PL=0
MOVL C00842 V=800.0 PL=0
MOVL C00843 V=800.0 PL=0
MOVL C00844 V=800.0 PL=0
MOVL C00845 V=800.0 PL=0
MOVL C00846 V=800.0 PL=0
MOVL C00847 V=800.0 PL=0
MOVL C00848 V=800.0 PL=0
MOVL C00849 V=800.0 PL=0
MOVL C00850 V=800.0 PL=0
MOVL C00851 V=800.0 PL=0
MOVL C00852 V=800.0 PL=0
MOVL C00853 V=800.0 PL=0
MOVL C00854 V=800.0 PL=0
MOVL C00855 V=800.0 PL=0
MOVL C00856 V=800.0 PL=0
MOVL C00857 V=800.0 PL=0
MOVL C00858 V=800.0 PL=0
MOVL C00859 V=800.0 PL=0
MOVL C00860 V=800.0 PL=0
MOVL C00861 V=800.0 PL=0
MOVL C00862 V=800.0 PL=0
MOVL C00863 V=800.0 PL=0
MOVL C00864 V=800.0 PL=0
MOVL C00865 V=800.0 PL=0
MOVL C00866 V=800.0 PL=0
MOVL C00867 V=800.0 PL=0
MOVL C00868 V=800.0 PL=0
MOVL C00869 V=800.0 PL=0
MOVL C00870 V=800.0 PL=0
MOVL C00871 V=800.0 PL=0
MOVL C00872 V=800.0 PL=0
MOVL C00873 V=800.0 PL=0
MOVL C00874 V=800.0 PL=0
MOVL C00875 V=800.0 PL=0
MOVL C00876 V=800.0 PL=0
MOVL C00877 V=800.0 PL=0
MOVL C00878 V=800.0 PL=0
MOVL C00879 V=800.0 PL=0
MOVL C00880 V=800.0 PL=0
MOVL C00881 V=800.0 PL=0
MOVL C00882 V=800.0 PL=0
MOVL C00883 V=800.0 PL=0
MOVL C00884 V=800.0 PL=0
MOVL C00885 V=800.0 PL=0
MOVL C00886 V=800.0 PL=0
MOVL C00887 V=800.0 PL=0
MOVL C00888 V=800.0 PL=0
MOVL C00889 V=800.0 PL=0
MOVL C00890 V=800.0 PL=0
MOVL C00891 V=800.0 PL=0
MOVL C00892 V=800.0 PL=0
MOVL C00893 V=800.0 PL=0
MOVL C00894 V=800.0 PL=0
MOVL C00895 V=800.0 PL=0
MOVL C00896 V=800.0 PL=0
MOVL C00897 V=800.0 PL=0
MOVL C00898 V=800.0 PL=0
MOVL C00899 V=800.0 PL=0
MOVL C00900 V=800.0 PL=0
MOVL C00901 V=800.0 PL=0
MOVL C00902 V=800.0 PL=0
MOVL C00903 V=800.0 PL=0
MOVL C00904 V=800.0 PL=0
MOVL C00905 V=800.0 PL=0
MOVL C00906 V=800.0 PL=0
MOVL C00907 V=800.0 PL=0
MOVL C00908 V=800.0 PL=0
MOVL C00909 V=800.0 PL=0
MOVL C00910 V=800.0 PL=0
MOVL C00911 V=800.0 PL=0
MOVL C00912 V=800.0 PL=0
MOVL C00913 V=800.0 PL=0
MOVL C00914 V=800.0 PL=0
MOVL C00915 V=800.0 PL=0
MOVL C00916 V=800.0 PL=0
MOVL C00917 V=800.0 PL=0
MOVL C00918 V=800.0 PL=0
MOVL C00919 V=800.0 PL=0
MOVL C00920 V=800.0 PL=0
MOVL C00921 V=800.0 PL=0
MOVL C00922 V=800.0 PL=0
MOVL C00923 V=800.0 PL=0
MOVL C00924 V=800.0 PL=0
MOVL C00925 V=800.0 PL=0
MOVL C00926 V=800.0 PL=0
MOVL C00927 V=800.0 PL=0
MOVL C00928 V=800.0 PL=0
MOVL C00929 V=800.0 PL=0
MOVL C00930 V=800.0 PL=0
MOVL C00931 V=800.0 PL=0
MOVL C00932 V=800.0 PL=0
MOVL C00933 V=800.0 PL=0
MOVL C00934 V=800.0 PL=0
MOVL C00935 V=800.0 PL=0
MOVL C00936 V=800.0 PL=0
MOVL C00937 V=800.0 PL=0
MOVL C00938 V=800.0 PL=0
MOVL C00939 V=800.0 PL=0
MOVL C00940 V=800.0 PL=0
MOVL C00941 V=800.0 PL=0
MOVL C00942 V=800.0 PL=0
MOVL C00943 V=800.0 PL=0
MOVL C00944 V=800.0 PL=0
MOVL C00945 V=800.0 PL=0
MOVL C00946 V=800.0 PL=0
MOVL C00947 V=800.0 PL=0
MOVL C00948 V=800.0 PL=0
MOVL C00949 V=800.0 PL=0
MOVL C00950 V=800.0 PL=0
MOVL C00951 V=800.0 PL=0
MOVL C00952 V=800.0 PL=0
MOVL C00953 V=800.0 PL=0
MOVL C00954 V=800.0 PL=0
MOVL C00955 V=800.0 PL=0
MOVL C00956 V=800.0 PL=0
MOVL C00957 V=800.0 PL=0
MOVL C00958 V=800.0 PL=0
MOVL C00959 V=800.0 PL=0
MOVL C00960 V=800.0 PL=0
MOVL C00961 V=800.0 PL=0
MOVL C00962 V=800.0 PL=0
MOVL C00963 V=800.0 PL=0
MOVL C00964 V=800.0 PL=0
MOVL C00965 V=800.0 PL=0
MOVL C00966 V=800.0 PL=0
MOVL C00967 V=800.0 PL=0
MOVL C00968 V=800.0 PL=0
MOVL C00969 V=800.0 PL=0
MOVL C00970 V=800.0 PL=0
MOVL C00971 V=800.0 PL=0
MOVL C00972 V=800.0 PL=0
MOVL C00973 V=800.0 PL=0
MOVL C00974 V=800.0 PL=0
MOVL C00975 V=800.0 PL=0
MOVL C00976 V=800.0 PL=0
MOVL C00977 V=800.0 PL=0
MOVL C00978 V=800.0 PL=0
MOVL C00979 V=800.0 PL=0
MOVL C00980 V=800.0 PL=0
MOVL C00981 V=800.0 PL=0
MOVL C00982 V=800.0 PL=0
MOVL C00983 V=800.0 PL=0
MOVL C00984 V=800.0 PL=0
MOVL C00985 V=800.0 PL=0
MOVL C00986 V=800.0 PL=0
MOVL C00987 V=800.0 PL=0
MOVL C00988 V=800.0 PL=0
MOVL C00989 V=800.0 PL=0
MOVL C00990 V=800.0 PL=0
MOVL C00991 V=800.0 PL=0
MOVL C00992 V=800.0 PL=0
MOVL C00993 V=800.0 PL=0
MOVL C00994 V=800.0 PL=0
MOVL C00995 V=800.0 PL=0
MOVL C00996 V=800.0 PL=0
MOVL C00997 V=800.0 PL=0
MOVL C00998 V=800.0 PL=0
MOVL C00999 V=800.0 PL=0
MOVL C01000 V=800.0 PL=0
MOVL C01001 V=800.0 PL=0
MOVL C01002 V=800.0 PL=0
MOVL C01003 V=800.0 PL=0
MOVL C01004 V=800.0 PL=0
MOVL C01005 V=800.0 PL=0
MOVL C01006 V=800.0 PL=0
MOVL C01007 V=800.0 PL=0
MOVL C01008 V=800.0 PL=0
MOVL C01009 V=800.0 PL=0
MOVL C01010 V=800.0 PL=0
MOVL C01011 V=800.0 PL=0
MOVL C01012 V=800.0 PL=0
MOVL C01013 V=800.0 PL=0
MOVL C01014 V=800.0 PL=0
MOVL C01015 V=800.0 PL=0
MOVL C01016 V=800.0 PL=0
MOVL C01017 V=800.0 PL=0
MOVL C01018 V=800.0 PL=0
MOVL C01019 V=800.0 PL=0
MOVL C01020 V=800.0 PL=0
MOVL C01021 V=800.0 PL=0
MOVL C01022 V=800.0 PL=0
MOVL C01023 V=800.0 PL=0
MOVL C01024 V=800.0 PL=0
MOVL C01025 V=800.0 PL=0
MOVL C01026 V=800.0 PL=0
MOVL C01027 V=800.0 PL=0
MOVL C01028 V=800.0 PL=0
MOVL C01029 V=800.0 PL=0
MOVL C01030 V=800.0 PL=0
MOVL C01031 V=800.0 PL=0
MOVL C01032 V=800.0 PL=0
MOVL C01033 V=800.0 PL=0
MOVL C01034 V=800.0 PL=0
MOVL C01035 V=800.0 PL=0
MOVL C01036 V=800.0 PL=0
MOVL C01037 V=800.0 PL=0
MOVL C01038 V=800.0 PL=0
MOVL C01039 V=800.0 PL=0
MOVL C01040 V=800.0 PL=0
MOVL C01041 V=800.0 PL=0
MOVL C01042 V=800.0 PL=0
MOVL C01043 V=800.0 PL=0
MOVL C01044 V=800.0 PL=0
MOVL C01045 V=800.0 PL=0
MOVL C01046 V=800.0 PL=0
MOVL C01047 V=800.0 PL=0
MOVL C01048 V=800.0 PL=0
MOVL C01049 V=800.0 PL=0
MOVL C01050 V=800.0 PL=0
MOVL C01051 V=800.0 PL=0
MOVL C01052 V=800.0 PL=0
MOVL C01053 V=800.0 PL=0
MOVL C01054 V=800.0 PL=0
MOVL C01055 V=800.0 PL=0
MOVL C01056 V=800.0 PL=0
MOVL C01057 V=800.0 PL=0
MOVL C01058 V=800.0 PL=0
MOVL C01059 V=800.0 PL=0
MOVL C01060 V=800.0 PL=0
MOVL C01061 V=800.0 PL=0
MOVL C01062 V=800.0 PL=0
MOVL C01063 V=800.0 PL=0
MOVL C01064 V=800.0 PL=0
MOVL C01065 V=800.0 PL=0
MOVL C01066 V=800.0 PL=0
MOVL C01067 V=800.0 PL=0
MOVL C01068 V=800.0 PL=0
MOVL C01069 V=800.0 PL=0
MOVL C01070 V=800.0 PL=0
MOVL C01071 V=800.0 PL=0
MOVL C01072 V=800.0 PL=0
MOVL C01073 V=800.0 PL=0
MOVL C01074 V=800.0 PL=0
MOVL C01075 V=800.0 PL=0
MOVL C01076 V=800.0 PL=0
MOVL C01077 V=800.0 PL=0
MOVL C01078 V=800.0 PL=0
MOVL C01079 V=800.0 PL=0
MOVL C01080 V=800.0 PL=0
MOVL C01081 V=800.0 PL=0
MOVL C01082 V=800.0 PL=0
MOVL C01083 V=800.0 PL=0
MOVL C01084 V=800.0 PL=0
MOVL C01085 V=800.0 PL=0
MOVL C01086 V=800.0 PL=0
MOVL C01087 V=800.0 PL=0
MOVL C01088 V=800.0 PL=0
MOVL C01089 V=800.0 PL=0
MOVL C01090 V=800.0 PL=0
MOVL C01091 V=800.0 PL=0
MOVL C01092 V=800.0 PL=0
MOVL C01093 V=800.0 PL=0
MOVL C01094 V=800.0 PL=0
MOVL C01095 V=800.0 PL=0
MOVL C01096 V=800.0 PL=0
MOVL C01097 V=800.0 PL=0
MOVL C01098 V=800.0 PL=0
MOVL C01099 V=800.0 PL=0
MOVL C01100 V=800.0 PL=0
MOVL C01101 V=800.0 PL=0
MOVL C01102 V=800.0 PL=0
MOVL C01103 V=800.0 PL=0
MOVL C01104 V=800.0 PL=0
MOVL C01105 V=800.0 PL=0
MOVL C01106 V=800.0 PL=0
MOVL C01107 V=800.0 PL=0
MOVL C01108 V=800.0 PL=0
MOVL C01109 V=800.0 PL=0
MOVL C01110 V=800.0 PL=0
MOVL C01111 V=800.0 PL=0
MOVL C01112 V=800.0 PL=0
MOVL C01113 V=800.0 PL=0
MOVL C01114 V=800.0 PL=0
MOVL C01115 V=800.0 PL=0
MOVL C01116 V=800.0 PL=0
MOVL C01117 V=800.0 PL=0
MOVL C01118 V=800.0 PL=0
MOVL C01119 V=800.0 PL=0
MOVL C01120 V=800.0 PL=0
MOVL C01121 V=800.0 PL=0
MOVL C01122 V=800.0 PL=0
MOVL C01123 V=800.0 PL=0
MOVL C01124 V=800.0 PL=0
MOVL C01125 V=800.0 PL=0
MOVL C01126 V=800.0 PL=0
MOVL C01127 V=800.0 PL=0
MOVL C01128 V=800.0 PL=0
MOVL C01129 V=800.0 PL=0
MOVL C01130 V=800.0 PL=0
MOVL C01131 V=800.0 PL=0
MOVL C01132 V=800.0 PL=0
MOVL C01133 V=800.0 PL=0
MOVL C01134 V=800.0 PL=0
MOVL C01135 V=800.0 PL=0
MOVL C01136 V=800.0 PL=0
MOVL C01137 V=800.0 PL=0
MOVL C01138 V=800.0 PL=0
MOVL C01139 V=800.0 PL=0
MOVL C01140 V=800.0 PL=0
MOVL C01141 V=800.0 PL=0
MOVL C01142 V=800.0 PL=0
MOVL C01143 V=800.0 PL=0
MOVL C01144 V=800.0 PL=0
MOVL C01145 V=800.0 PL=0
MOVL C01146 V=800.0 PL=0
MOVL C01147 V=800.0 PL=0
MOVL C01148 V=800.0 PL=0
MOVL C01149 V=800.0 PL=0
MOVL C01150 V=800.0 PL=0
MOVL C01151 V=800.0 PL=0
MOVL C01152 V=800.0 PL=0
MOVL C01153 V=800.0 PL=0
MOVL C01154 V=800.0 PL=0
MOVL C01155 V=800.0 PL=0
MOVL C01156 V=800.0 PL=0
MOVL C01157 V=800.0 PL=0
MOVL C01158 V=800.0 PL=0
MOVL C01159 V=800.0 PL=0
MOVL C01160 V=800.0 PL=0
MOVL C01161 V=800.0 PL=0
MOVL C01162 V=800.0 PL=0
MOVL C01163 V=800.0 PL=0
MOVL C01164 V=800.0 PL=0
MOVL C01165 V=800.0 PL=0
MOVL C01166 V=800.0 PL=0
MOVL C01167 V=800.0 PL=0
MOVL C01168 V=800.0 PL=0
MOVL C01169 V=800.0 PL=0
MOVL C01170 V=800.0 PL=0
MOVL C01171 V=800.0 PL=0
MOVL C01172 V=800.0 PL=0
MOVL C01173 V=800.0 PL=0
MOVL C01174 V=800.0 PL=0
MOVL C01175 V=800.0 PL=0
MOVL C01176 V=800.0 PL=0
MOVL C01177 V=800.0 PL=0
MOVL C01178 V=800.0 PL=0
MOVL C01179 V=800.0 PL=0
MOVL C01180 V=800.0 PL=0
MOVL C01181 V=800.0 PL=0
MOVL C01182 V=800.0 PL=0
MOVL C01183 V=800.0 PL=0
MOVL C01184 V=800.0 PL=0
MOVL C01185 V=800.0 PL=0
MOVL C01186 V=800.0 PL=0
MOVL C01187 V=800.0 PL=0
MOVL C01188 V=800.0 PL=0
MOVL C01189 V=800.0 PL=0
MOVL C01190 V=800.0 PL=0
MOVL C01191 V=800.0 PL=0
MOVL C01192 V=800.0 PL=0
MOVL C01193 V=800.0 PL=0
MOVL C01194 V=800.0 PL=0
MOVL C01195 V=800.0 PL=0
MOVL C01196 V=800.0 PL=0
MOVL C01197 V=800.0 PL=0
MOVL C01198 V=800.0 PL=0
MOVL C01199 V=800.0 PL=0
MOVL C01200 V=800.0 PL=0
MOVL C01201 V=800.0 PL=0
MOVL C01202 V=800.0 PL=0
MOVL C01203 V=800.0 PL=0
MOVL C01204 V=800.0 PL=0
MOVL C01205 V=800.0 PL=0
MOVL C01206 V=800.0 PL=0
MOVL C01207 V=800.0 PL=0
MOVL C01208 V=800.0 PL=0
MOVL C01209 V=800.0 PL=0
MOVL C01210 V=800.0 PL=0
MOVL C01211 V=800.0 PL=0
MOVL C01212 V=800.0 PL=0
MOVL C01213 V=800.0 PL=0
MOVL C01214 V=800.0 PL=0
MOVL C01215 V=800.0 PL=0
MOVL C01216 V=800.0 PL=0
MOVL C01217 V=800.0 PL=0
MOVL C01218 V=800.0 PL=0
MOVL C01219 V=800.0 PL=0
MOVL C01220 V=800.0 PL=0
MOVL C01221 V=800.0 PL=0
MOVL C01222 V=800.0 PL=0
MOVL C01223 V=800.0 PL=0
MOVL C01224 V=800.0 PL=0
MOVL C01225 V=800.0 PL=0
MOVL C01226 V=800.0 PL=0
MOVL C01227 V=800.0 PL=0
MOVL C01228 V=800.0 PL=0
MOVL C01229 V=800.0 PL=0
MOVL C01230 V=800.0 PL=0
MOVL C01231 V=800.0 PL=0
MOVL C01232 V=800.0 PL=0
MOVL C01233 V=800.0 PL=0
MOVL C01234 V=800.0 PL=0
MOVL C01235 V=800.0 PL=0
MOVL C01236 V=800.0 PL=0
MOVL C01237 V=800.0 PL=0
MOVL C01238 V=800.0 PL=0
MOVL C01239 V=800.0 PL=0
MOVL C01240 V=800.0 PL=0
MOVL C01241 V=800.0 PL=0
MOVL C01242 V=800.0 PL=0
MOVL C01243 V=800.0 PL=0
MOVL C01244 V=800.0 PL=0
MOVL C01245 V=800.0 PL=0
MOVL C01246 V=800.0 PL=0
MOVL C01247 V=800.0 PL=0
MOVL C01248 V=800.0 PL=0
MOVL C01249 V=800.0 PL=0
MOVL C01250 V=800.0 PL=0
MOVL C01251 V=800.0 PL=0
MOVL C01252 V=800.0 PL=0
MOVL C01253 V=800.0 PL=0
MOVL C01254 V=800.0 PL=0
MOVL C01255 V=800.0 PL=0
MOVL C01256 V=800.0 PL=0
MOVL C01257 V=800.0 PL=0
MOVL C01258 V=800.0 PL=0
MOVL C01259 V=800.0 PL=0
MOVL C01260 V=800.0 PL=0
MOVL C01261 V=800.0 PL=0
MOVL C01262 V=800.0 PL=0
MOVL C01263 V=800.0 PL=0
MOVL C01264 V=800.0 PL=0
MOVL C01265 V=800.0 PL=0
MOVL C01266 V=800.0 PL=0
MOVL C01267 V=800.0 PL=0
MOVL C01268 V=800.0 PL=0
MOVL C01269 V=800.0 PL=0
MOVL C01270 V=800.0 PL=0
MOVL C01271 V=800.0 PL=0
MOVL C01272 V=800.0 PL=0
MOVL C01273 V=800.0 PL=0
MOVL C01274 V=800.0 PL=0
MOVL C01275 V=800.0 PL=0
MOVL C01276 V=800.0 PL=0
MOVL C01277 V=800.0 PL=0
MOVL C01278 V=800.0 PL=0
MOVL C01279 V=800.0 PL=0
MOVL C01280 V=800.0 PL=0
MOVL C01281 V=800.0 PL=0
MOVL C01282 V=800.0 PL=0
MOVL C01283 V=800.0 PL=0
MOVL C01284 V=800.0 PL=0
MOVL C01285 V=800.0 PL=0
MOVL C01286 V=800.0 PL=0
MOVL C01287 V=800.0 PL=0
MOVL C01288 V=800.0 PL=0
MOVL C01289 V=800.0 PL=0
MOVL C01290 V=800.0 PL=0
MOVL C01291 V=800.0 PL=0
MOVL C01292 V=800.0 PL=0
MOVL C01293 V=800.0 PL=0
MOVL C01294 V=800.0 PL=0
MOVL C01295 V=800.0 PL=0
MOVL C01296 V=800.0 PL=0
MOVL C01297 V=800.0 PL=0
MOVL C01298 V=800.0 PL=0
MOVL C01299 V=800.0 PL=0
MOVL C01300 V=800.0 PL=0
MOVL C01301 V=800.0 PL=0
MOVL C01302 V=800.0 PL=0
MOVL C01303 V=800.0 PL=0
MOVL C01304 V=800.0 PL=0
MOVL C01305 V=800.0 PL=0
MOVL C01306 V=800.0 PL=0
MOVL C01307 V=800.0 PL=0
MOVL C01308 V=800.0 PL=0
MOVL C01309 V=800.0 PL=0
MOVL C01310 V=800.0 PL=0
MOVL C01311 V=800.0 PL=0
MOVL C01312 V=800.0 PL=0
MOVL C01313 V=800.0 PL=0
MOVL C01314 V=800.0 PL=0
MOVL C01315 V=800.0 PL=0
MOVL C01316 V=800.0 PL=0
MOVL C01317 V=800.0 PL=0
MOVL C01318 V=800.0 PL=0
MOVL C01319 V=800.0 PL=0
MOVL C01320 V=800.0 PL=0
MOVL C01321 V=800.0 PL=0
MOVL C01322 V=800.0 PL=0
MOVL C01323 V=800.0 PL=0
MOVL C01324 V=800.0 PL=0
MOVL C01325 V=800.0 PL=0
MOVL C01326 V=800.0 PL=0
MOVL C01327 V=800.0 PL=0
MOVL C01328 V=800.0 PL=0
MOVL C01329 V=800.0 PL=0
MOVL C01330 V=800.0 PL=0
MOVL C01331 V=800.0 PL=0
MOVL C01332 V=800.0 PL=0
MOVL C01333 V=800.0 PL=0
MOVL C01334 V=800.0 PL=0
MOVL C01335 V=800.0 PL=0
MOVL C01336 V=800.0 PL=0
MOVL C01337 V=800.0 PL=0
MOVL C01338 V=800.0 PL=0
MOVL C01339 V=800.0 PL=0
MOVL C01340 V=800.0 PL=0
MOVL C01341 V=800.0 PL=0
MOVL C01342 V=800.0 PL=0
MOVL C01343 V=800.0 PL=0
MOVL C01344 V=800.0 PL=0
MOVL C01345 V=800.0 PL=0
MOVL C01346 V=800.0 PL=0
MOVL C01347 V=800.0 PL=0
MOVL C01348 V=800.0 PL=0
MOVL C01349 V=800.0 PL=0
MOVL C01350 V=800.0 PL=0
MOVL C01351 V=800.0 PL=0
MOVL C01352 V=800.0 PL=0
MOVL C01353 V=800.0 PL=0
MOVL C01354 V=800.0 PL=0
MOVL C01355 V=800.0 PL=0
MOVL C01356 V=800.0 PL=0
MOVL C01357 V=800.0 PL=0
MOVL C01358 V=800.0 PL=0
MOVL C01359 V=800.0 PL=0
MOVL C01360 V=800.0 PL=0
MOVL C01361 V=800.0 PL=0
MOVL C01362 V=800.0 PL=0
MOVL C01363 V=800.0 PL=0
MOVL C01364 V=800.0 PL=0
MOVL C01365 V=800.0 PL=0
MOVL C01366 V=800.0 PL=0
MOVL C01367 V=800.0 PL=0
MOVL C01368 V=800.0 PL=0
MOVL C01369 V=800.0 PL=0
MOVL C01370 V=800.0 PL=0
MOVL C01371 V=800.0 PL=0
MOVL C01372 V=800.0 PL=0
MOVL C01373 V=800.0 PL=0
MOVL C01374 V=800.0 PL=0
MOVL C01375 V=800.0 PL=0
MOVL C01376 V=800.0 PL=0
MOVL C01377 V=800.0 PL=0
MOVL C01378 V=800.0 PL=0
MOVL C01379 V=800.0 PL=0
MOVL C01380 V=800.0 PL=0
MOVL C01381 V=800.0 PL=0
MOVL C01382 V=800.0 PL=0
MOVL C01383 V=800.0 PL=0
MOVL C01384 V=800.0 PL=0
MOVL C01385 V=800.0 PL=0
MOVL C01386 V=800.0 PL=0
MOVL C01387 V=800.0 PL=0
MOVL C01388 V=800.0 PL=0
MOVL C01389 V=800.0 PL=0
MOVL C01390 V=800.0 PL=0
MOVL C01391 V=800.0 PL=0
MOVL C01392 V=800.0 PL=0
MOVL C01393 V=800.0 PL=0
MOVL C01394 V=800.0 PL=0
MOVL C01395 V=800.0 PL=0
MOVL C01396 V=800.0 PL=0
MOVL C01397 V=800.0 PL=0
MOVL C01398 V=800.0 PL=0
MOVL C01399 V=800.0 PL=0
MOVL C01400 V=800.0 PL=0
MOVL C01401 V=800.0 PL=0
MOVL C01402 V=800.0 PL=0
MOVL C01403 V=800.0 PL=0
MOVL C01404 V=800.0 PL=0
MOVL C01405 V=800.0 PL=0
MOVL C01406 V=800.0 PL=0
MOVL C01407 V=800.0 PL=0
MOVL C01408 V=800.0 PL=0
MOVL C01409 V=800.0 PL=0
MOVL C01410 V=800.0 PL=0
MOVL C01411 V=800.0 PL=0
MOVL C01412 V=800.0 PL=0
MOVL C01413 V=800.0 PL=0
MOVL C01414 V=800.0 PL=0
MOVL C01415 V=800.0 PL=0
MOVL C01416 V=800.0 PL=0
MOVL C01417 V=800.0 PL=0
MOVL C01418 V=800.0 PL=0
MOVL C01419 V=800.0 PL=0
MOVL C01420 V=800.0 PL=0
MOVL C01421 V=800.0 PL=0
MOVL C01422 V=800.0 PL=0
MOVL C01423 V=800.0 PL=0
MOVL C01424 V=800.0 PL=0
MOVL C01425 V=800.0 PL=0
MOVL C01426 V=800.0 PL=0
MOVL C01427 V=800.0 PL=0
MOVL C01428 V=800.0 PL=0
MOVL C01429 V=800.0 PL=0
MOVL C01430 V=800.0 PL=0
MOVL C01431 V=800.0 PL=0
MOVL C01432 V=800.0 PL=0
MOVL C01433 V=800.0 PL=0
MOVL C01434 V=800.0 PL=0
MOVL C01435 V=800.0 PL=0
MOVL C01436 V=800.0 PL=0
MOVL C01437 V=800.0 PL=0
MOVL C01438 V=800.0 PL=0
MOVL C01439 V=800.0 PL=0
MOVL C01440 V=800.0 PL=0
MOVL C01441 V=800.0 PL=0
MOVL C01442 V=800.0 PL=0
MOVL C01443 V=800.0 PL=0
MOVL C01444 V=800.0 PL=0
MOVL C01445 V=800.0 PL=0
MOVL C01446 V=800.0 PL=0
MOVL C01447 V=800.0 PL=0
MOVL C01448 V=800.0 PL=0
MOVL C01449 V=800.0 PL=0
MOVL C01450 V=800.0 PL=0
MOVL C01451 V=800.0 PL=0
MOVL C01452 V=800.0 PL=0
MOVL C01453 V=800.0 PL=0
MOVL C01454 V=800.0 PL=0
MOVL C01455 V=800.0 PL=0
MOVL C01456 V=800.0 PL=0
MOVL C01457 V=800.0 PL=0
MOVL C01458 V=800.0 PL=0
MOVL C01459 V=800.0 PL=0
MOVL C01460 V=800.0 PL=0
MOVL C01461 V=800.0 PL=0
MOVL C01462 V=800.0 PL=0
MOVL C01463 V=800.0 PL=0
MOVL C01464 V=800.0 PL=0
MOVL C01465 V=800.0 PL=0
MOVL C01466 V=800.0 PL=0
MOVL C01467 V=800.0 PL=0
MOVL C01468 V=800.0 PL=0
MOVL C01469 V=800.0 PL=0
MOVL C01470 V=800.0 PL=0
MOVL C01471 V=800.0 PL=0
MOVL C01472 V=800.0 PL=0
MOVL C01473 V=800.0 PL=0
MOVL C01474 V=800.0 PL=0
MOVL C01475 V=800.0 PL=0
MOVL C01476 V=800.0 PL=0
MOVL C01477 V=800.0 PL=0
MOVL C01478 V=800.0 PL=0
MOVL C01479 V=800.0 PL=0
MOVL C01480 V=800.0 PL=0
MOVL C01481 V=800.0 PL=0
MOVL C01482 V=800.0 PL=0
MOVL C01483 V=800.0 PL=0
MOVL C01484 V=800.0 PL=0
MOVL C01485 V=800.0 PL=0
MOVL C01486 V=800.0 PL=0
MOVL C01487 V=800.0 PL=0
MOVL C01488 V=800.0 PL=0
MOVL C01489 V=800.0 PL=0
MOVL C01490 V=800.0 PL=0
MOVL C01491 V=800.0 PL=0
MOVL C01492 V=800.0 PL=0
MOVL C01493 V=800.0 PL=0
MOVL C01494 V=800.0 PL=0
MOVL C01495 V=800.0 PL=0
MOVL C01496 V=800.0 PL=0
MOVL C01497 V=800.0 PL=0
MOVL C01498 V=800.0 PL=0
MOVL C01499 V=800.0 PL=0
MOVL C01500 V=800.0 PL=0
MOVL C01501 V=800.0 PL=0
MOVL C01502 V=800.0 PL=0
MOVL C01503 V=800.0 PL=0
MOVL C01504 V=800.0 PL=0
MOVL C01505 V=800.0 PL=0
MOVL C01506 V=800.0 PL=0
MOVL C01507 V=800.0 PL=0
MOVL C01508 V=800.0 PL=0
MOVL C01509 V=800.0 PL=0
MOVL C01510 V=800.0 PL=0
MOVL C01511 V=800.0 PL=0
MOVL C01512 V=800.0 PL=0
MOVL C01513 V=800.0 PL=0
MOVL C01514 V=800.0 PL=0
MOVL C01515 V=800.0 PL=0
MOVL C01516 V=800.0 PL=0
MOVL C01517 V=800.0 PL=0
MOVL C01518 V=800.0 PL=0
MOVL C01519 V=800.0 PL=0
MOVL C01520 V=800.0 PL=0
MOVL C01521 V=800.0 PL=0
MOVL C01522 V=800.0 PL=0
MOVL C01523 V=800.0 PL=0
MOVL C01524 V=800.0 PL=0
MOVL C01525 V=800.0 PL=0
MOVL C01526 V=800.0 PL=0
MOVL C01527 V=800.0 PL=0
MOVL C01528 V=800.0 PL=0
MOVL C01529 V=800.0 PL=0
MOVL C01530 V=800.0 PL=0
MOVL C01531 V=800.0 PL=0
MOVL C01532 V=800.0 PL=0
MOVL C01533 V=800.0 PL=0
MOVL C01534 V=800.0 PL=0
MOVL C01535 V=800.0 PL=0
MOVL C01536 V=800.0 PL=0
MOVL C01537 V=800.0 PL=0
MOVL C01538 V=800.0 PL=0
MOVL C01539 V=800.0 PL=0
MOVL C01540 V=800.0 PL=0
MOVL C01541 V=800.0 PL=0
MOVL C01542 V=800.0 PL=0
MOVL C01543 V=800.0 PL=0
MOVL C01544 V=800.0 PL=0
MOVL C01545 V=800.0 PL=0
MOVL C01546 V=800.0 PL=0
MOVL C01547 V=800.0 PL=0
MOVL C01548 V=800.0 PL=0
MOVL C01549 V=800.0 PL=0
MOVL C01550 V=800.0 PL=0
MOVL C01551 V=800.0 PL=0
MOVL C01552 V=800.0 PL=0
MOVL C01553 V=800.0 PL=0
MOVL C01554 V=800.0 PL=0
MOVL C01555 V=800.0 PL=0
MOVL C01556 V=800.0 PL=0
MOVL C01557 V=800.0 PL=0
MOVL C01558 V=800.0 PL=0
MOVL C01559 V=800.0 PL=0
MOVL C01560 V=800.0 PL=0
MOVL C01561 V=800.0 PL=0
MOVL C01562 V=800.0 PL=0
MOVL C01563 V=800.0 PL=0
MOVL C01564 V=800.0 PL=0
MOVL C01565 V=800.0 PL=0
MOVL C01566 V=800.0 PL=0
MOVL C01567 V=800.0 PL=0
MOVL C01568 V=800.0 PL=0
MOVL C01569 V=800.0 PL=0
MOVL C01570 V=800.0 PL=0
MOVL C01571 V=800.0 PL=0
MOVL C01572 V=800.0 PL=0
MOVL C01573 V=800.0 PL=0
MOVL C01574 V=800.0 PL=0
MOVL C01575 V=800.0 PL=0
MOVL C01576 V=800.0 PL=0
MOVL C01577 V=800.0 PL=0
MOVL C01578 V=800.0 PL=0
MOVL C01579 V=800.0 PL=0
MOVL C01580 V=800.0 PL=0
MOVL C01581 V=800.0 PL=0
MOVL C01582 V=800.0 PL=0
MOVL C01583 V=800.0 PL=0
MOVL C01584 V=800.0 PL=0
MOVL C01585 V=800.0 PL=0
MOVL C01586 V=800.0 PL=0
MOVL C01587 V=800.0 PL=0
MOVL C01588 V=800.0 PL=0
MOVL C01589 V=800.0 PL=0
MOVL C01590 V=800.0 PL=0
MOVL C01591 V=800.0 PL=0
MOVL C01592 V=800.0 PL=0
MOVL C01593 V=800.0 PL=0
MOVL C01594 V=800.0 PL=0
MOVL C01595 V=800.0 PL=0
MOVL C01596 V=800.0 PL=0
MOVL C01597 V=800.0 PL=0
MOVL C01598 V=800.0 PL=0
MOVL C01599 V=800.0 PL=0
MOVL C01600 V=800.0 PL=0
MOVL C01601 V=800.0 PL=0
MOVL C01602 V=800.0 PL=0
MOVL C01603 V=800.0 PL=0
MOVL C01604 V=800.0 PL=0
MOVL C01605 V=800.0 PL=0
MOVL C01606 V=800.0 PL=0
MOVL C01607 V=800.0 PL=0
MOVL C01608 V=800.0 PL=0
MOVL C01609 V=800.0 PL=0
MOVL C01610 V=800.0 PL=0
MOVL C01611 V=800.0 PL=0
MOVL C01612 V=800.0 PL=0
MOVL C01613 V=800.0 PL=0
MOVL C01614 V=800.0 PL=0
MOVL C01615 V=800.0 PL=0
MOVL C01616 V=800.0 PL=0
MOVL C01617 V=800.0 PL=0
MOVL C01618 V=800.0 PL=0
MOVL C01619 V=800.0 PL=0
MOVL C01620 V=800.0 PL=0
MOVL C01621 V=800.0 PL=0
MOVL C01622 V=800.0 PL=0
MOVL C01623 V=800.0 PL=0
MOVL C01624 V=800.0 PL=0
MOVL C01625 V=800.0 PL=0
MOVL C01626 V=800.0 PL=0
MOVL C01627 V=800.0 PL=0
MOVL C01628 V=800.0 PL=0
MOVL C01629 V=800.0 PL=0
MOVL C01630 V=800.0 PL=0
MOVL C01631 V=800.0 PL=0
MOVL C01632 V=800.0 PL=0
MOVL C01633 V=800.0 PL=0
MOVL C01634 V=800.0 PL=0
MOVL C01635 V=800.0 PL=0
MOVL C01636 V=800.0 PL=0
MOVL C01637 V=800.0 PL=0
MOVL C01638 V=800.0 PL=0
MOVL C01639 V=800.0 PL=0
MOVL C01640 V=800.0 PL=0
MOVL C01641 V=800.0 PL=0
MOVL C01642 V=800.0 PL=0
MOVL C01643 V=800.0 PL=0
MOVL C01644 V=800.0 PL=0
MOVL C01645 V=800.0 PL=0
MOVL C01646 V=800.0 PL=0
MOVL C01647 V=800.0 PL=0
MOVL C01648 V=800.0 PL=0
MOVL C01649 V=800.0 PL=0
MOVL C01650 V=800.0 PL=0
MOVL C01651 V=800.0 PL=0
MOVL C01652 V=800.0 PL=0
MOVL C01653 V=800.0 PL=0
MOVL C01654 V=800.0 PL=0
MOVL C01655 V=800.0 PL=0
MOVL C01656 V=800.0 PL=0
MOVL C01657 V=800.0 PL=0
MOVL C01658 V=800.0 PL=0
MOVL C01659 V=800.0 PL=0
MOVL C01660 V=800.0 PL=0
MOVL C01661 V=800.0 PL=0
MOVL C01662 V=800.0 PL=0
MOVL C01663 V=800.0 PL=0
MOVL C01664 V=800.0 PL=0
MOVL C01665 V=800.0 PL=0
MOVL C01666 V=800.0 PL=0
MOVL C01667 V=800.0 PL=0
MOVL C01668 V=800.0 PL=0
MOVL C01669 V=800.0 PL=0
MOVL C01670 V=800.0 PL=0
MOVL C01671 V=800.0 PL=0
MOVL C01672 V=800.0 PL=0
MOVL C01673 V=800.0 PL=0
MOVL C01674 V=800.0 PL=0
MOVL C01675 V=800.0 PL=0
MOVL C01676 V=800.0 PL=0
MOVL C01677 V=800.0 PL=0
MOVL C01678 V=800.0 PL=0
MOVL C01679 V=800.0 PL=0
MOVL C01680 V=800.0 PL=0
MOVL C01681 V=800.0 PL=0
MOVL C01682 V=800.0 PL=0
MOVL C01683 V=800.0 PL=0
MOVL C01684 V=800.0 PL=0
MOVL C01685 V=800.0 PL=0
MOVL C01686 V=800.0 PL=0
MOVL C01687 V=800.0 PL=0
MOVL C01688 V=800.0 PL=0
MOVL C01689 V=800.0 PL=0
MOVL C01690 V=800.0 PL=0
MOVL C01691 V=800.0 PL=0
MOVL C01692 V=800.0 PL=0
MOVL C01693 V=800.0 PL=0
MOVL C01694 V=800.0 PL=0
MOVL C01695 V=800.0 PL=0
MOVL C01696 V=800.0 PL=0
MOVL C01697 V=800.0 PL=0
MOVL C01698 V=800.0 PL=0
MOVL C01699 V=800.0 PL=0
MOVL C01700 V=800.0 PL=0
MOVL C01701 V=800.0 PL=0
MOVL C01702 V=800.0 PL=0
MOVL C01703 V=800.0 PL=0
MOVL C01704 V=800.0 PL=0
MOVL C01705 V=800.0 PL=0
MOVL C01706 V=800.0 PL=0
MOVL C01707 V=800.0 PL=0
MOVL C01708 V=800.0 PL=0
MOVL C01709 V=800.0 PL=0
MOVL C01710 V=800.0 PL=0
MOVL C01711 V=800.0 PL=0
MOVL C01712 V=800.0 PL=0
MOVL C01713 V=800.0 PL=0
MOVL C01714 V=800.0 PL=0
MOVL C01715 V=800.0 PL=0
MOVL C01716 V=800.0 PL=0
MOVL C01717 V=800.0 PL=0
MOVL C01718 V=800.0 PL=0
MOVL C01719 V=800.0 PL=0
MOVL C01720 V=800.0 PL=0
MOVL C01721 V=800.0 PL=0
MOVL C01722 V=800.0 PL=0
MOVL C01723 V=800.0 PL=0
MOVL C01724 V=800.0 PL=0
MOVL C01725 V=800.0 PL=0
MOVL C01726 V=800.0 PL=0
MOVL C01727 V=800.0 PL=0
MOVL C01728 V=800.0 PL=0
MOVL C01729 V=800.0 PL=0
MOVL C01730 V=800.0 PL=0
MOVL C01731 V=800.0 PL=0
MOVL C01732 V=800.0 PL=0
MOVL C01733 V=800.0 PL=0
MOVL C01734 V=800.0 PL=0
MOVL C01735 V=800.0 PL=0
MOVL C01736 V=800.0 PL=0
MOVL C01737 V=800.0 PL=0
MOVL C01738 V=800.0 PL=0
MOVL C01739 V=800.0 PL=0
MOVL C01740 V=800.0 PL=0
MOVL C01741 V=800.0 PL=0
MOVL C01742 V=800.0 PL=0
MOVL C01743 V=800.0 PL=0
MOVL C01744 V=800.0 PL=0
MOVL C01745 V=800.0 PL=0
MOVL C01746 V=800.0 PL=0
MOVL C01747 V=800.0 PL=0
MOVL C01748 V=800.0 PL=0
MOVL C01749 V=800.0 PL=0
MOVL C01750 V=800.0 PL=0
MOVL C01751 V=800.0 PL=0
MOVL C01752 V=800.0 PL=0
MOVL C01753 V=800.0 PL=0
MOVL C01754 V=800.0 PL=0
MOVL C01755 V=800.0 PL=0
MOVL C01756 V=800.0 PL=0
MOVL C01757 V=800.0 PL=0
MOVL C01758 V=800.0 PL=0
MOVL C01759 V=800.0 PL=0
MOVL C01760 V=800.0 PL=0
MOVL C01761 V=800.0 PL=0
MOVL C01762 V=800.0 PL=0
MOVL C01763 V=800.0 PL=0
MOVL C01764 V=800.0 PL=0
MOVL C01765 V=800.0 PL=0
MOVL C01766 V=800.0 PL=0
MOVL C01767 V=800.0 PL=0
MOVL C01768 V=800.0 PL=0
MOVL C01769 V=800.0 PL=0
MOVL C01770 V=800.0 PL=0
MOVL C01771 V=800.0 PL=0
MOVL C01772 V=800.0 PL=0
MOVL C01773 V=800.0 PL=0
MOVL C01774 V=800.0 PL=0
MOVL C01775 V=800.0 PL=0
MOVL C01776 V=800.0 PL=0
MOVL C01777 V=800.0 PL=0
MOVL C01778 V=800.0 PL=0
MOVL C01779 V=800.0 PL=0
MOVL C01780 V=800.0 PL=0
MOVL C01781 V=800.0 PL=0
MOVL C01782 V=800.0 PL=0
MOVL C01783 V=800.0 PL=0
MOVL C01784 V=800.0 PL=0
MOVL C01785 V=800.0 PL=0
MOVL C01786 V=800.0 PL=0
MOVL C01787 V=800.0 PL=0
MOVL C01788 V=800.0 PL=0
MOVL C01789 V=800.0 PL=0
MOVL C01790 V=800.0 PL=0
MOVL C01791 V=800.0 PL=0
MOVL C01792 V=800.0 PL=0
MOVL C01793 V=800.0 PL=0
MOVL C01794 V=800.0 PL=0
MOVL C01795 V=800.0 PL=0
MOVL C01796 V=800.0 PL=0
MOVL C01797 V=800.0 PL=0
MOVL C01798 V=800.0 PL=0
MOVL C01799 V=800.0 PL=0
MOVL C01800 V=800.0 PL=0
MOVL C01801 V=800.0 PL=0
MOVL C01802 V=800.0 PL=0
MOVL C01803 V=800.0 PL=0
MOVL C01804 V=800.0 PL=0
MOVL C01805 V=800.0 PL=0
MOVL C01806 V=800.0 PL=0
MOVL C01807 V=800.0 PL=0
MOVL C01808 V=800.0 PL=0
MOVL C01809 V=800.0 PL=0
MOVL C01810 V=800.0 PL=0
MOVL C01811 V=800.0 PL=0
MOVL C01812 V=800.0 PL=0
MOVL C01813 V=800.0 PL=0
MOVL C01814 V=800.0 PL=0
MOVL C01815 V=800.0 PL=0
MOVL C01816 V=800.0 PL=0
MOVL C01817 V=800.0 PL=0
MOVL C01818 V=800.0 PL=0
MOVL C01819 V=800.0 PL=0
MOVL C01820 V=800.0 PL=0
MOVL C01821 V=800.0 PL=0
MOVL C01822 V=800.0 PL=0
MOVL C01823 V=800.0 PL=0
MOVL C01824 V=800.0 PL=0
MOVL C01825 V=800.0 PL=0
MOVL C01826 V=800.0 PL=0
MOVL C01827 V=800.0 PL=0
MOVL C01828 V=800.0 PL=0
MOVL C01829 V=800.0 PL=0
MOVL C01830 V=800.0 PL=0
MOVL C01831 V=800.0 PL=0
MOVL C01832 V=800.0 PL=0
MOVL C01833 V=800.0 PL=0
MOVL C01834 V=800.0 PL=0
MOVL C01835 V=800.0 PL=0
MOVL C01836 V=800.0 PL=0
MOVL C01837 V=800.0 PL=0
MOVL C01838 V=800.0 PL=0
MOVL C01839 V=800.0 PL=0
MOVL C01840 V=800.0 PL=0
MOVL C01841 V=800.0 PL=0
MOVL C01842 V=800.0 PL=0
MOVL C01843 V=800.0 PL=0
MOVL C01844 V=800.0 PL=0
MOVL C01845 V=800.0 PL=0
MOVL C01846 V=800.0 PL=0
MOVL C01847 V=800.0 PL=0
MOVL C01848 V=800.0 PL=0
MOVL C01849 V=800.0 PL=0
MOVL C01850 V=800.0 PL=0
MOVL C01851 V=800.0 PL=0
MOVL C01852 V=800.0 PL=0
MOVL C01853 V=800.0 PL=0
MOVL C01854 V=800.0 PL=0
MOVL C01855 V=800.0 PL=0
MOVL C01856 V=800.0 PL=0
MOVL C01857 V=800.0 PL=0
MOVL C01858 V=800.0 PL=0
MOVL C01859 V=800.0 PL=0
MOVL C01860 V=800.0 PL=0
MOVL C01861 V=800.0 PL=0
MOVL C01862 V=800.0 PL=0
MOVL C01863 V=800.0 PL=0
MOVL C01864 V=800.0 PL=0
MOVL C01865 V=800.0 PL=0
MOVL C01866 V=800.0 PL=0
MOVL C01867 V=800.0 PL=0
MOVL C01868 V=800.0 PL=0
MOVL C01869 V=800.0 PL=0
MOVL C01870 V=800.0 PL=0
MOVL C01871 V=800.0 PL=0
MOVL C01872 V=800.0 PL=0
MOVL C01873 V=800.0 PL=0
MOVL C01874 V=800.0 PL=0
MOVL C01875 V=800.0 PL=0
MOVL C01876 V=800.0 PL=0
MOVL C01877 V=800.0 PL=0
MOVL C01878 V=800.0 PL=0
MOVL C01879 V=800.0 PL=0
MOVL C01880 V=800.0 PL=0
MOVL C01881 V=800.0 PL=0
MOVL C01882 V=800.0 PL=0
MOVL C01883 V=800.0 PL=0
MOVL C01884 V=800.0 PL=0
MOVL C01885 V=800.0 PL=0
MOVL C01886 V=800.0 PL=0
MOVL C01887 V=800.0 PL=0
MOVL C01888 V=800.0 PL=0
MOVL C01889 V=800.0 PL=0
MOVL C01890 V=800.0 PL=0
MOVL C01891 V=800.0 PL=0
MOVL C01892 V=800.0 PL=0
MOVL C01893 V=800.0 PL=0
MOVL C01894 V=800.0 PL=0
MOVL C01895 V=800.0 PL=0
MOVL C01896 V=800.0 PL=0
MOVL C01897 V=800.0 PL=0
MOVL C01898 V=800.0 PL=0
MOVL C01899 V=800.0 PL=0
MOVL C01900 V=800.0 PL=0
MOVL C01901 V=800.0 PL=0
MOVL C01902 V=800.0 PL=0
MOVL C01903 V=800.0 PL=0
MOVL C01904 V=800.0 PL=0
MOVL C01905 V=800.0 PL=0
MOVL C01906 V=800.0 PL=0
MOVL C01907 V=800.0 PL=0
MOVL C01908 V=800.0 PL=0
MOVL C01909 V=800.0 PL=0
MOVL C01910 V=800.0 PL=0
MOVL C01911 V=800.0 PL=0
MOVL C01912 V=800.0 PL=0
MOVL C01913 V=800.0 PL=0
MOVL C01914 V=800.0 PL=0
MOVL C01915 V=800.0 PL=0
MOVL C01916 V=800.0 PL=0
MOVL C01917 V=800.0 PL=0
MOVL C01918 V=800.0 PL=0
MOVL C01919 V=800.0 PL=0
MOVL C01920 V=800.0 PL=0
MOVL C01921 V=800.0 PL=0
MOVL C01922 V=800.0 PL=0
MOVL C01923 V=800.0 PL=0
MOVL C01924 V=800.0 PL=0
MOVL C01925 V=800.0 PL=0
MOVL C01926 V=800.0 PL=0
MOVL C01927 V=800.0 PL=0
MOVL C01928 V=800.0 PL=0
MOVL C01929 V=800.0 PL=0
MOVL C01930 V=800.0 PL=0
MOVL C01931 V=800.0 PL=0
MOVL C01932 V=800.0 PL=0
MOVL C01933 V=800.0 PL=0
MOVL C01934 V=800.0 PL=0
MOVL C01935 V=800.0 PL=0
MOVL C01936 V=800.0 PL=0
MOVL C01937 V=800.0 PL=0
MOVL C01938 V=800.0 PL=0
MOVL C01939 V=800.0 PL=0
MOVL C01940 V=800.0 PL=0
MOVL C01941 V=800.0 PL=0
MOVL C01942 V=800.0 PL=0
MOVL C01943 V=800.0 PL=0
MOVL C01944 V=800.0 PL=0
MOVL C01945 V=800.0 PL=0
MOVL C01946 V=800.0 PL=0
MOVL C01947 V=800.0 PL=0
MOVL C01948 V=800.0 PL=0
MOVL C01949 V=800.0 PL=0
MOVL C01950 V=800.0 PL=0
MOVL C01951 V=800.0 PL=0
MOVL C01952 V=800.0 PL=0
MOVL C01953 V=800.0 PL=0
MOVL C01954 V=800.0 PL=0
MOVL C01955 V=800.0 PL=0
MOVL C01956 V=800.0 PL=0
MOVL C01957 V=800.0 PL=0
MOVL C01958 V=800.0 PL=0
MOVL C01959 V=800.0 PL=0
MOVL C01960 V=800.0 PL=0
MOVL C01961 V=800.0 PL=0
MOVL C01962 V=800.0 PL=0
MOVL C01963 V=800.0 PL=0
MOVL C01964 V=800.0 PL=0
MOVL C01965 V=800.0 PL=0
MOVL C01966 V=800.0 PL=0
MOVL C01967 V=800.0 PL=0
MOVL C01968 V=800.0 PL=0
MOVL C01969 V=800.0 PL=0
MOVL C01970 V=800.0 PL=0
MOVL C01971 V=800.0 PL=0
MOVL C01972 V=800.0 PL=0
MOVL C01973 V=800.0 PL=0
MOVL C01974 V=800.0 PL=0
MOVL C01975 V=800.0 PL=0
MOVL C01976 V=800.0 PL=0
MOVL C01977 V=800.0 PL=0
MOVL C01978 V=800.0 PL=0
MOVL C01979 V=800.0 PL=0
MOVL C01980 V=800.0 PL=0
MOVL C01981 V=800.0 PL=0
MOVL C01982 V=800.0 PL=0
MOVL C01983 V=800.0 PL=0
MOVL C01984 V=800.0 PL=0
MOVL C01985 V=800.0 PL=0
MOVL C01986 V=800.0 PL=0
MOVL C01987 V=800.0 PL=0
MOVL C01988 V=800.0 PL=0
MOVL C01989 V=800.0 PL=0
MOVL C01990 V=800.0 PL=0
MOVL C01991 V=800.0 PL=0
MOVL C01992 V=800.0 PL=0
MOVL C01993 V=800.0 PL=0
MOVL C01994 V=800.0 PL=0
MOVL C01995 V=800.0 PL=0
MOVL C01996 V=800.0 PL=0
MOVL C01997 V=800.0 PL=0
MOVL C01998 V=800.0 PL=0
MOVL C01999 V=800.0 PL=0
MOVL C02000 V=800.0 PL=0
MOVL C02001 V=800.0 PL=0
MOVL C02002 V=800.0 PL=0
MOVL C02003 V=800.0 PL=0
MOVL C02004 V=800.0 PL=0
MOVL C02005 V=800.0 PL=0
MOVL C02006 V=800.0 PL=0
MOVL C02007 V=800.0 PL=0
MOVL C02008 V=800.0 PL=0
MOVL C02009 V=800.0 PL=0
MOVL C02010 V=800.0 PL=0
MOVL C02011 V=800.0 PL=0
MOVL C02012 V=800.0 PL=0
MOVL C02013 V=800.0 PL=0
MOVL C02014 V=800.0 PL=0
MOVL C02015 V=800.0 PL=0
MOVL C02016 V=800.0 PL=0
MOVL C02017 V=800.0 PL=0
MOVL C02018 V=800.0 PL=0
MOVL C02019 V=800.0 PL=0
MOVL C02020 V=800.0 PL=0
MOVL C02021 V=800.0 PL=0
MOVL C02022 V=800.0 PL=0
MOVL C02023 V=800.0 PL=0
MOVL C02024 V=800.0 PL=0
MOVL C02025 V=800.0 PL=0
MOVL C02026 V=800.0 PL=0
MOVL C02027 V=800.0 PL=0
MOVL C02028 V=800.0 PL=0
MOVL C02029 V=800.0 PL=0
MOVL C02030 V=800.0 PL=0
MOVL C02031 V=800.0 PL=0
MOVL C02032 V=800.0 PL=0
MOVL C02033 V=800.0 PL=0
MOVL C02034 V=800.0 PL=0
MOVL C02035 V=800.0 PL=0
MOVL C02036 V=800.0 PL=0
MOVL C02037 V=800.0 PL=0
MOVL C02038 V=800.0 PL=0
MOVL C02039 V=800.0 PL=0
MOVL C02040 V=800.0 PL=0
MOVL C02041 V=800.0 PL=0
MOVL C02042 V=800.0 PL=0
MOVL C02043 V=800.0 PL=0
MOVL C02044 V=800.0 PL=0
MOVL C02045 V=800.0 PL=0
MOVL C02046 V=800.0 PL=0
MOVL C02047 V=800.0 PL=0
MOVL C02048 V=800.0 PL=0
MOVL C02049 V=800.0 PL=0
MOVL C02050 V=800.0 PL=0
MOVL C02051 V=800.0 PL=0
MOVL C02052 V=800.0 PL=0
MOVL C02053 V=800.0 PL=0
MOVL C02054 V=800.0 PL=0
MOVL C02055 V=800.0 PL=0
MOVL C02056 V=800.0 PL=0
MOVL C02057 V=800.0 PL=0
MOVL C02058 V=800.0 PL=0
MOVL C02059 V=800.0 PL=0
MOVL C02060 V=800.0 PL=0
MOVL C02061 V=800.0 PL=0
MOVL C02062 V=800.0 PL=0
MOVL C02063 V=800.0 PL=0
MOVL C02064 V=800.0 PL=0
MOVL C02065 V=800.0 PL=0
MOVL C02066 V=800.0 PL=0
MOVL C02067 V=800.0 PL=0
MOVL C02068 V=800.0 PL=0
MOVL C02069 V=800.0 PL=0
MOVL C02070 V=800.0 PL=0
MOVL C02071 V=800.0 PL=0
MOVL C02072 V=800.0 PL=0
MOVL C02073 V=800.0 PL=0
MOVL C02074 V=800.0 PL=0
MOVL C02075 V=800.0 PL=0
MOVL C02076 V=800.0 PL=0
MOVL C02077 V=800.0 PL=0
MOVL C02078 V=800.0 PL=0
MOVL C02079 V=800.0 PL=0
MOVL C02080 V=800.0 PL=0
MOVL C02081 V=800.0 PL=0
MOVL C02082 V=800.0 PL=0
MOVL C02083 V=800.0 PL=0
